Universal Robots PolyScope program: marco_robot_test.urp

Program marco_robot_test (installation=default directory=/programs createdIn=5.11.9.1010452 lastSavedIn=5.11.9.1010452 robotSerialNumber=20225200364)
Calibrated DH parameters: a=[0.00002, -0.569483, -0.54992, -0.00001, -0.000036, 0]; d=[0.180894, -146.691669, 192.918669, -46.053088, 0.119778, 0.115602]; alpha=[1.571425, -0.001534, 0.003359, 1.568739, -1.571477, 0]; deltaTheta=[0, 0.376258, -0.101074, -0.275185, -0.000002, 0]
Robot Program (runOnlyOnce=true)
  Script file /programs/usbdisk/marco_robot_5.script
    | def Machining3():
    |   # Default parameters:
    |   global speed_ms = 0.3
    |   global speed_rads = 0.75
    |   global accel_mss = 3
    |   global accel_radss = 1.2
    |   global blend_radius_m = 0.001
    | 
    |   # Add subprograms here
    |   # Start of main program
    |   # Program generated by RoboDK v5.6.5 for UR10e on 17/10/2023 12:20:24
    |   # Using nominal kinematics.
    |   blend_radius_m = 0.001
    |   speed_ms = 1.000
    |   # set_reference(p[0.335000, -0.154000, -0.002000, 0.000000, 0.000000, 0.000000])
    |   set_tcp(p[0.000000, 0.000000, 0.252000, 0.000000, 0.000000, 0.000000])
    |   # Show Tool
    |   movej([0.089160, -1.181798, -2.545827, -0.984764, 1.570796, 1.659956],accel_radss,speed_rads,0,blend_radius_m)
    |   movel([0.089160, -1.275562, -2.606033, -0.830794, 1.570796, 1.659956],accel_mss,speed_ms,0,blend_radius_m)
    |   speed_ms = 0.005
    |   movel([0.089160, -1.286495, -2.611612, -0.814282, 1.570796, 1.659956],accel_mss,speed_ms,0,blend_radius_m)
    |   movel([0.089160, -1.309264, -2.622500, -0.780625, 1.570796, 1.659956],accel_mss,speed_ms,0,blend_radius_m)
    |   movel([0.083541, -1.305906, -2.624527, -0.781955, 1.570796, 1.654337],accel_mss,speed_ms,0,blend_radius_m)
    |   movel([0.089160, -1.309264, -2.622500, -0.780625, 1.570796, 1.659956],accel_mss,speed_ms,0,blend_radius_m)
    |   movel([0.089160, -1.286495, -2.611612, -0.814282, 1.570796, 1.659956],accel_mss,speed_ms,0,blend_radius_m)
    |   movel([0.081204, -1.281682, -2.614420, -0.816287, 1.570796, 1.652001],accel_mss,speed_ms,0,blend_radius_m)
    |   movel([0.081204, -1.304518, -2.625361, -0.782510, 1.570796, 1.652001],accel_mss,speed_ms,0,blend_radius_m)
    |   movel([0.098719, -1.298708, -2.628824, -0.784857, 1.570796, 1.669516],accel_mss,speed_ms,0,blend_radius_m)
    |   movel([0.097011, -1.314060, -2.619578, -0.778751, 1.570796, 1.667807],accel_mss,speed_ms,0,blend_radius_m)
    |   movel([0.079808, -1.319640, -2.616140, -0.776609, 1.570796, 1.650604],accel_mss,speed_ms,0,blend_radius_m)
    |   movel([0.081204, -1.304518, -2.625361, -0.782510, 1.570796, 1.652001],accel_mss,speed_ms,0,blend_radius_m)
    |   movel([0.098719, -1.298708, -2.628824, -0.784857, 1.570796, 1.669516],accel_mss,speed_ms,0,blend_radius_m)
    |   movel([0.097011, -1.314060, -2.619578, -0.778751, 1.570796, 1.667807],accel_mss,speed_ms,0,blend_radius_m)
    |   movel([0.079808, -1.319640, -2.616140, -0.776609, 1.570796, 1.650604],accel_mss,speed_ms,0,blend_radius_m)
    |   movel([0.081204, -1.304518, -2.625361, -0.782510, 1.570796, 1.652001],accel_mss,speed_ms,0,blend_radius_m)
    |   movel([0.081204, -1.281682, -2.614420, -0.816287, 1.570796, 1.652001],accel_mss,speed_ms,0,blend_radius_m)
    |   movel([0.077108, -1.278531, -2.616242, -0.817615, 1.570796, 1.647904],accel_mss,speed_ms,0,blend_radius_m)
    |   movel([0.077108, -1.301410, -2.627219, -0.783760, 1.570796, 1.647904],accel_mss,speed_ms,0,blend_radius_m)
    |   movel([0.055264, -1.309051, -2.622629, -0.780709, 1.570796, 1.626060],accel_mss,speed_ms,0,blend_radius_m)
    |   movel([0.054551, -1.320244, -2.615765, -0.776379, 1.570796, 1.625347],accel_mss,speed_ms,0,blend_radius_m)
    |   movel([0.076104, -1.312829, -2.620331, -0.779229, 1.570796, 1.646901],accel_mss,speed_ms,0,blend_radius_m)
    |   movel([0.054551, -1.320244, -2.615765, -0.776379, 1.570796, 1.625347],accel_mss,speed_ms,0,blend_radius_m)
    |   movel([0.055264, -1.309051, -2.622629, -0.780709, 1.570796, 1.626060],accel_mss,speed_ms,0,blend_radius_m)
    |   movel([0.077108, -1.301410, -2.627219, -0.783760, 1.570796, 1.647904],accel_mss,speed_ms,0,blend_radius_m)
    |   movel([0.077108, -1.278531, -2.616242, -0.817615, 1.570796, 1.647904],accel_mss,speed_ms,0,blend_radius_m)
    |   movel([0.074534, -1.291116, -2.608888, -0.812385, 1.570796, 1.645331],accel_mss,speed_ms,0,blend_radius_m)
    |   movel([0.074534, -1.313820, -2.619725, -0.778844, 1.570796, 1.645331],accel_mss,speed_ms,0,blend_radius_m)
    |   movel([0.056039, -1.320179, -2.615806, -0.776404, 1.570796, 1.626835],accel_mss,speed_ms,0,blend_radius_m)
    |   movel([0.074534, -1.313820, -2.619725, -0.778844, 1.570796, 1.645331],accel_mss,speed_ms,0,blend_radius_m)
    |   movel([0.074534, -1.291116, -2.608888, -0.812385, 1.570796, 1.645331],accel_mss,speed_ms,0,blend_radius_m)
    |   movel([0.055828, -1.300854, -2.603061, -0.808474, 1.570796, 1.626625],accel_mss,speed_ms,0,blend_radius_m)
    |   movel([0.055828, -1.323418, -2.613789, -0.775182, 1.570796, 1.626625],accel_mss,speed_ms,0,blend_radius_m)
    |   movel([0.074252, -1.317114, -2.617702, -0.777573, 1.570796, 1.645049],accel_mss,speed_ms,0,blend_radius_m)
    |   movel([0.055828, -1.323418, -2.613789, -0.775182, 1.570796, 1.626625],accel_mss,speed_ms,0,blend_radius_m)
    |   movel([0.055828, -1.300854, -2.603061, -0.808474, 1.570796, 1.626625],accel_mss,speed_ms,0,blend_radius_m)
    |   movel([0.075501, -1.297125, -2.605307, -0.809958, 1.570796, 1.646297],accel_mss,speed_ms,0,blend_radius_m)
    |   movel([0.075501, -1.319743, -2.616077, -0.776570, 1.570796, 1.646297],accel_mss,speed_ms,0,blend_radius_m)
    |   movel([0.054122, -1.327025, -2.611526, -0.773837, 1.570796, 1.624918],accel_mss,speed_ms,0,blend_radius_m)
    |   movel([0.052635, -1.350841, -2.596143, -0.765405, 1.570796, 1.623432],accel_mss,speed_ms,0,blend_radius_m)
    |   movel([0.073235, -1.346070, -2.599287, -0.767032, 1.570796, 1.644031],accel_mss,speed_ms,0,blend_radius_m)
    |   movel([0.052635, -1.350841, -2.596143, -0.765405, 1.570796, 1.623432],accel_mss,speed_ms,0,blend_radius_m)
    |   movel([0.054122, -1.327025, -2.611526, -0.773837, 1.570796, 1.624918],accel_mss,speed_ms,0,blend_radius_m)
    |   movel([0.075501, -1.319743, -2.616077, -0.776570, 1.570796, 1.646297],accel_mss,speed_ms,0,blend_radius_m)
    |   movel([0.075501, -1.297125, -2.605307, -0.809958, 1.570796, 1.646297],accel_mss,speed_ms,0,blend_radius_m)
    |   movel([0.084967, -1.313702, -2.595186, -0.803501, 1.570796, 1.655763],accel_mss,speed_ms,0,blend_radius_m)
    |   movel([0.084967, -1.336075, -2.605773, -0.770542, 1.570796, 1.655763],accel_mss,speed_ms,0,blend_radius_m)
    |   movel([0.126975, -1.323371, -2.613818, -0.775199, 1.570796, 1.697771],accel_mss,speed_ms,0,blend_radius_m)
    |   movel([0.124703, -1.339286, -2.603704, -0.769399, 1.570796, 1.695499],accel_mss,speed_ms,0,blend_radius_m)
    |   movel([0.083467, -1.351474, -2.595724, -0.765192, 1.570796, 1.654263],accel_mss,speed_ms,0,blend_radius_m)
    |   movel([0.084967, -1.336075, -2.605773, -0.770542, 1.570796, 1.655763],accel_mss,speed_ms,0,blend_radius_m)
    |   movel([0.126975, -1.323371, -2.613818, -0.775199, 1.570796, 1.697771],accel_mss,speed_ms,0,blend_radius_m)
    |   movel([0.124703, -1.339286, -2.603704, -0.769399, 1.570796, 1.695499],accel_mss,speed_ms,0,blend_radius_m)
    |   movel([0.083467, -1.351474, -2.595724, -0.765192, 1.570796, 1.654263],accel_mss,speed_ms,0,blend_radius_m)
    |   movel([0.084967, -1.336075, -2.605773, -0.770542, 1.570796, 1.655763],accel_mss,speed_ms,0,blend_radius_m)
    |   movel([0.084967, -1.313702, -2.595186, -0.803501, 1.570796, 1.655763],accel_mss,speed_ms,0,blend_radius_m)
    |   movel([0.093012, -1.328943, -2.585565, -0.797880, 1.570796, 1.663809],accel_mss,speed_ms,0,blend_radius_m)
    |   movel([0.093012, -1.351081, -2.595984, -0.765324, 1.570796, 1.663809],accel_mss,speed_ms,0,blend_radius_m)
    |   movel([0.114947, -1.344626, -2.600233, -0.767530, 1.570796, 1.685744],accel_mss,speed_ms,0,blend_radius_m)
    |   movel([0.114417, -1.348663, -2.597583, -0.766144, 1.570796, 1.685214],accel_mss,speed_ms,0,blend_radius_m)
    |   movel([0.092587, -1.355051, -2.593343, -0.763996, 1.570796, 1.663383],accel_mss,speed_ms,0,blend_radius_m)
    |   movel([0.093012, -1.351081, -2.595984, -0.765324, 1.570796, 1.663809],accel_mss,speed_ms,0,blend_radius_m)
    |   movel([0.114947, -1.344626, -2.600233, -0.767530, 1.570796, 1.685744],accel_mss,speed_ms,0,blend_radius_m)
    |   movel([0.114417, -1.348663, -2.597583, -0.766144, 1.570796, 1.685214],accel_mss,speed_ms,0,blend_radius_m)
    |   movel([0.092587, -1.355051, -2.593343, -0.763996, 1.570796, 1.663383],accel_mss,speed_ms,0,blend_radius_m)
    |   movel([0.093012, -1.351081, -2.595984, -0.765324, 1.570796, 1.663809],accel_mss,speed_ms,0,blend_radius_m)
    |   movel([0.093012, -1.328943, -2.585565, -0.797880, 1.570796, 1.663809],accel_mss,speed_ms,0,blend_radius_m)
    |   movel([0.097348, -1.351902, -2.570489, -0.789998, 1.570796, 1.668144],accel_mss,speed_ms,0,blend_radius_m)
    |   movel([0.097348, -1.373670, -2.580657, -0.758062, 1.570796, 1.668144],accel_mss,speed_ms,0,blend_radius_m)
    |   movel([0.101037, -1.372618, -2.581387, -0.758385, 1.570796, 1.671834],accel_mss,speed_ms,0,blend_radius_m)
    |   movel([0.104717, -1.371577, -2.582107, -0.758705, 1.570796, 1.675514],accel_mss,speed_ms,0,blend_radius_m)
    |   movel([0.100259, -1.379284, -2.576735, -0.756370, 1.570796, 1.671055],accel_mss,speed_ms,0,blend_radius_m)
    |   movel([0.097348, -1.373670, -2.580657, -0.758062, 1.570796, 1.668144],accel_mss,speed_ms,0,blend_radius_m)
    |   movel([0.101037, -1.372618, -2.581387, -0.758385, 1.570796, 1.671834],accel_mss,speed_ms,0,blend_radius_m)
    |   movel([0.104717, -1.371577, -2.582107, -0.758705, 1.570796, 1.675514],accel_mss,speed_ms,0,blend_radius_m)
    |   movel([0.100259, -1.379284, -2.576735, -0.756370, 1.570796, 1.671055],accel_mss,speed_ms,0,blend_radius_m)
    |   movel([0.097348, -1.373670, -2.580657, -0.758062, 1.570796, 1.668144],accel_mss,speed_ms,0,blend_radius_m)
    |   movel([0.097348, -1.351902, -2.570489, -0.789998, 1.570796, 1.668144],accel_mss,speed_ms,0,blend_radius_m)
    |   movel([0.088027, -1.372703, -2.556208, -0.783478, 1.570796, 1.658823],accel_mss,speed_ms,0,blend_radius_m)
    |   movel([0.088027, -1.394119, -2.566152, -0.752118, 1.570796, 1.658823],accel_mss,speed_ms,0,blend_radius_m)
    |   movel([0.109776, -1.388105, -2.570480, -0.753803, 1.570796, 1.680572],accel_mss,speed_ms,0,blend_radius_m)
    |   movel([0.109257, -1.392184, -2.567551, -0.752654, 1.570796, 1.680053],accel_mss,speed_ms,0,blend_radius_m)
    |   movel([0.087614, -1.398134, -2.563233, -0.751022, 1.570796, 1.658410],accel_mss,speed_ms,0,blend_radius_m)
    |   movel([0.088027, -1.394119, -2.566152, -0.752118, 1.570796, 1.658823],accel_mss,speed_ms,0,blend_radius_m)
    |   movel([0.109776, -1.388105, -2.570480, -0.753803, 1.570796, 1.680572],accel_mss,speed_ms,0,blend_radius_m)
    |   movel([0.109257, -1.392184, -2.567551, -0.752654, 1.570796, 1.680053],accel_mss,speed_ms,0,blend_radius_m)
    |   movel([0.087614, -1.398134, -2.563233, -0.751022, 1.570796, 1.658410],accel_mss,speed_ms,0,blend_radius_m)
    |   movel([0.088027, -1.394119, -2.566152, -0.752118, 1.570796, 1.658823],accel_mss,speed_ms,0,blend_radius_m)
    |   movel([0.088027, -1.372703, -2.556208, -0.783478, 1.570796, 1.658823],accel_mss,speed_ms,0,blend_radius_m)
    |   movel([0.137771, -1.304245, -2.601003, -0.807141, 1.570796, 1.708567],accel_mss,speed_ms,0,blend_radius_m)
    |   movel([0.137771, -1.326759, -2.611694, -0.773936, 1.570796, 1.708567],accel_mss,speed_ms,0,blend_radius_m)
    |   movel([0.159338, -1.318850, -2.616630, -0.776910, 1.570796, 1.730135],accel_mss,speed_ms,0,blend_radius_m)
    |   movel([0.164004, -1.292855, -2.632269, -0.787265, 1.570796, 1.734800],accel_mss,speed_ms,0,blend_radius_m)
    |   movel([0.142128, -1.298999, -2.628652, -0.784738, 1.570796, 1.712924],accel_mss,speed_ms,0,blend_radius_m)
    |   movel([0.164004, -1.292855, -2.632269, -0.787265, 1.570796, 1.734800],accel_mss,speed_ms,0,blend_radius_m)
    |   movel([0.159338, -1.318850, -2.616630, -0.776910, 1.570796, 1.730135],accel_mss,speed_ms,0,blend_radius_m)
    |   movel([0.137771, -1.326759, -2.611694, -0.773936, 1.570796, 1.708567],accel_mss,speed_ms,0,blend_radius_m)
    |   movel([0.137771, -1.304245, -2.601003, -0.807141, 1.570796, 1.708567],accel_mss,speed_ms,0,blend_radius_m)
    |   movel([0.144204, -1.272270, -2.619828, -0.820291, 1.570796, 1.715001],accel_mss,speed_ms,0,blend_radius_m)
    |   movel([0.144204, -1.295233, -2.630875, -0.786282, 1.570796, 1.715001],accel_mss,speed_ms,0,blend_radius_m)
    |   movel([0.163060, -1.289910, -2.633985, -0.788494, 1.570796, 1.733856],accel_mss,speed_ms,0,blend_radius_m)
    |   movel([0.144204, -1.295233, -2.630875, -0.786282, 1.570796, 1.715001],accel_mss,speed_ms,0,blend_radius_m)
    |   movel([0.144204, -1.272270, -2.619828, -0.820291, 1.570796, 1.715001],accel_mss,speed_ms,0,blend_radius_m)
    |   movel([0.143289, -1.268681, -2.621861, -0.821846, 1.570796, 1.714086],accel_mss,speed_ms,0,blend_radius_m)
    |   movel([0.143289, -1.291691, -2.632948, -0.787749, 1.570796, 1.714086],accel_mss,speed_ms,0,blend_radius_m)
    |   movel([0.165352, -1.285426, -2.636577, -0.790386, 1.570796, 1.736149],accel_mss,speed_ms,0,blend_radius_m)
    |   movel([0.167598, -1.273136, -2.643552, -0.795701, 1.570796, 1.738395],accel_mss,speed_ms,0,blend_radius_m)
    |   movel([0.145223, -1.279606, -2.639904, -0.792879, 1.570796, 1.716019],accel_mss,speed_ms,0,blend_radius_m)
    |   movel([0.167598, -1.273136, -2.643552, -0.795701, 1.570796, 1.738395],accel_mss,speed_ms,0,blend_radius_m)
    |   movel([0.165352, -1.285426, -2.636577, -0.790386, 1.570796, 1.736149],accel_mss,speed_ms,0,blend_radius_m)
    |   movel([0.143289, -1.291691, -2.632948, -0.787749, 1.570796, 1.714086],accel_mss,speed_ms,0,blend_radius_m)
    |   movel([0.143289, -1.268681, -2.621861, -0.821846, 1.570796, 1.714086],accel_mss,speed_ms,0,blend_radius_m)
    |   movel([0.144765, -1.268733, -2.621832, -0.821824, 1.570796, 1.715562],accel_mss,speed_ms,0,blend_radius_m)
    |   movel([0.144765, -1.291742, -2.632919, -0.787728, 1.570796, 1.715562],accel_mss,speed_ms,0,blend_radius_m)
    |   movel([0.163697, -1.286370, -2.636034, -0.789985, 1.570796, 1.734494],accel_mss,speed_ms,0,blend_radius_m)
    |   movel([0.144765, -1.291742, -2.632919, -0.787728, 1.570796, 1.715562],accel_mss,speed_ms,0,blend_radius_m)
    |   movel([0.144765, -1.268733, -2.621832, -0.821824, 1.570796, 1.715562],accel_mss,speed_ms,0,blend_radius_m)
    |   movel([0.125413, -1.167058, -2.673236, -0.872095, 1.570796, 1.696210],accel_mss,speed_ms,0,blend_radius_m)
    |   movel([0.125413, -1.191107, -2.685463, -0.835818, 1.570796, 1.696210],accel_mss,speed_ms,0,blend_radius_m)
    |   movel([0.125706, -1.190153, -2.685906, -0.836330, 1.570796, 1.696503],accel_mss,speed_ms,0,blend_radius_m)
    |   movel([0.127514, -1.187943, -2.686927, -0.837519, 1.570796, 1.698310],accel_mss,speed_ms,0,blend_radius_m)
    |   movel([0.128757, -1.187262, -2.687241, -0.837886, 1.570796, 1.699553],accel_mss,speed_ms,0,blend_radius_m)
    |   movel([0.159607, -1.176201, -2.692265, -0.843923, 1.570796, 1.730403],accel_mss,speed_ms,0,blend_radius_m)
    |   movel([0.160858, -1.176036, -2.692339, -0.844014, 1.570796, 1.731655],accel_mss,speed_ms,0,blend_radius_m)
    |   movel([0.162120, -1.177291, -2.691776, -0.843322, 1.570796, 1.732916],accel_mss,speed_ms,0,blend_radius_m)
    |   movel([0.162101, -1.178007, -2.691454, -0.842928, 1.570796, 1.732898],accel_mss,speed_ms,0,blend_radius_m)
    |   movel([0.160218, -1.189028, -2.686427, -0.836935, 1.570796, 1.731014],accel_mss,speed_ms,0,blend_radius_m)
    |   movel([0.159776, -1.190238, -2.685867, -0.836284, 1.570796, 1.730573],accel_mss,speed_ms,0,blend_radius_m)
    |   movel([0.158190, -1.192057, -2.685022, -0.835310, 1.570796, 1.728986],accel_mss,speed_ms,0,blend_radius_m)
    |   movel([0.156814, -1.192816, -2.684669, -0.834905, 1.570796, 1.727611],accel_mss,speed_ms,0,blend_radius_m)
    |   movel([0.126529, -1.203419, -2.679664, -0.829306, 1.570796, 1.697325],accel_mss,speed_ms,0,blend_radius_m)
    |   movel([0.125786, -1.203591, -2.679582, -0.829216, 1.570796, 1.696582],accel_mss,speed_ms,0,blend_radius_m)
    |   movel([0.124122, -1.202858, -2.679932, -0.829599, 1.570796, 1.694918],accel_mss,speed_ms,0,blend_radius_m)
    |   movel([0.123975, -1.201767, -2.680452, -0.830170, 1.570796, 1.694771],accel_mss,speed_ms,0,blend_radius_m)
    |   movel([0.125413, -1.191107, -2.685463, -0.835818, 1.570796, 1.696210],accel_mss,speed_ms,0,blend_radius_m)
    |   movel([0.125706, -1.190153, -2.685906, -0.836330, 1.570796, 1.696503],accel_mss,speed_ms,0,blend_radius_m)
    |   movel([0.127514, -1.187943, -2.686927, -0.837519, 1.570796, 1.698310],accel_mss,speed_ms,0,blend_radius_m)
    |   movel([0.128757, -1.187262, -2.687241, -0.837886, 1.570796, 1.699553],accel_mss,speed_ms,0,blend_radius_m)
    |   movel([0.159607, -1.176201, -2.692265, -0.843923, 1.570796, 1.730403],accel_mss,speed_ms,0,blend_radius_m)
    |   movel([0.160858, -1.176036, -2.692339, -0.844014, 1.570796, 1.731655],accel_mss,speed_ms,0,blend_radius_m)
    |   movel([0.162120, -1.177291, -2.691776, -0.843322, 1.570796, 1.732916],accel_mss,speed_ms,0,blend_radius_m)
    |   movel([0.162101, -1.178007, -2.691454, -0.842928, 1.570796, 1.732898],accel_mss,speed_ms,0,blend_radius_m)
    |   movel([0.160218, -1.189028, -2.686427, -0.836935, 1.570796, 1.731014],accel_mss,speed_ms,0,blend_radius_m)
    |   movel([0.159776, -1.190238, -2.685867, -0.836284, 1.570796, 1.730573],accel_mss,speed_ms,0,blend_radius_m)
    |   movel([0.158190, -1.192057, -2.685022, -0.835310, 1.570796, 1.728986],accel_mss,speed_ms,0,blend_radius_m)
    |   movel([0.156814, -1.192816, -2.684669, -0.834905, 1.570796, 1.727611],accel_mss,speed_ms,0,blend_radius_m)
    |   movel([0.126529, -1.203419, -2.679664, -0.829306, 1.570796, 1.697325],accel_mss,speed_ms,0,blend_radius_m)
    |   movel([0.125786, -1.203591, -2.679582, -0.829216, 1.570796, 1.696582],accel_mss,speed_ms,0,blend_radius_m)
    |   movel([0.124122, -1.202858, -2.679932, -0.829599, 1.570796, 1.694918],accel_mss,speed_ms,0,blend_radius_m)
    |   movel([0.123975, -1.201767, -2.680452, -0.830170, 1.570796, 1.694771],accel_mss,speed_ms,0,blend_radius_m)
    |   movel([0.125413, -1.191107, -2.685463, -0.835818, 1.570796, 1.696210],accel_mss,speed_ms,0,blend_radius_m)
    |   movel([0.125413, -1.167058, -2.673236, -0.872095, 1.570796, 1.696210],accel_mss,speed_ms,0,blend_radius_m)
    |   movel([0.123336, -1.182593, -2.666121, -0.863674, 1.570796, 1.694132],accel_mss,speed_ms,0,blend_radius_m)
    |   movel([0.123336, -1.206525, -2.678175, -0.827689, 1.570796, 1.694132],accel_mss,speed_ms,0,blend_radius_m)
    |   movel([0.159381, -1.193945, -2.684142, -0.834303, 1.570796, 1.730178],accel_mss,speed_ms,0,blend_radius_m)
    |   movel([0.154982, -1.220061, -2.671558, -0.820770, 1.570796, 1.725778],accel_mss,speed_ms,0,blend_radius_m)
    |   movel([0.119973, -1.231829, -2.665636, -0.814924, 1.570796, 1.690769],accel_mss,speed_ms,0,blend_radius_m)
    |   movel([0.123336, -1.206525, -2.678175, -0.827689, 1.570796, 1.694132],accel_mss,speed_ms,0,blend_radius_m)
    |   movel([0.159381, -1.193945, -2.684142, -0.834303, 1.570796, 1.730178],accel_mss,speed_ms,0,blend_radius_m)
    |   movel([0.154982, -1.220061, -2.671558, -0.820770, 1.570796, 1.725778],accel_mss,speed_ms,0,blend_radius_m)
    |   movel([0.119973, -1.231829, -2.665636, -0.814924, 1.570796, 1.690769],accel_mss,speed_ms,0,blend_radius_m)
    |   movel([0.123336, -1.206525, -2.678175, -0.827689, 1.570796, 1.694132],accel_mss,speed_ms,0,blend_radius_m)
    |   movel([0.123336, -1.182593, -2.666121, -0.863674, 1.570796, 1.694132],accel_mss,speed_ms,0,blend_radius_m)
    |   movel([0.122335, -1.208273, -2.653796, -0.850320, 1.570796, 1.693131],accel_mss,speed_ms,0,blend_radius_m)
    |   movel([0.122335, -1.231976, -2.665561, -0.814852, 1.570796, 1.693131],accel_mss,speed_ms,0,blend_radius_m)
    |   movel([0.151945, -1.222034, -2.670576, -0.819779, 1.570796, 1.722741],accel_mss,speed_ms,0,blend_radius_m)
    |   movel([0.153970, -1.222028, -2.670579, -0.819782, 1.570796, 1.724766],accel_mss,speed_ms,0,blend_radius_m)
    |   movel([0.154423, -1.223410, -2.669889, -0.819090, 1.570796, 1.725219],accel_mss,speed_ms,0,blend_radius_m)
    |   movel([0.153408, -1.225329, -2.668927, -0.818133, 1.570796, 1.724204],accel_mss,speed_ms,0,blend_radius_m)
    |   movel([0.151526, -1.226585, -2.668295, -0.817510, 1.570796, 1.722322],accel_mss,speed_ms,0,blend_radius_m)
    |   movel([0.121726, -1.236519, -2.663231, -0.812639, 1.570796, 1.692523],accel_mss,speed_ms,0,blend_radius_m)
    |   movel([0.120074, -1.236452, -2.663266, -0.812672, 1.570796, 1.690871],accel_mss,speed_ms,0,blend_radius_m)
    |   movel([0.119542, -1.235104, -2.663959, -0.813326, 1.570796, 1.690338],accel_mss,speed_ms,0,blend_radius_m)
    |   movel([0.120485, -1.233242, -2.664914, -0.814233, 1.570796, 1.691281],accel_mss,speed_ms,0,blend_radius_m)
    |   movel([0.122335, -1.231976, -2.665561, -0.814852, 1.570796, 1.693131],accel_mss,speed_ms,0,blend_radius_m)
    |   movel([0.151945, -1.222034, -2.670576, -0.819779, 1.570796, 1.722741],accel_mss,speed_ms,0,blend_radius_m)
    |   movel([0.153970, -1.222028, -2.670579, -0.819782, 1.570796, 1.724766],accel_mss,speed_ms,0,blend_radius_m)
    |   movel([0.154423, -1.223410, -2.669889, -0.819090, 1.570796, 1.725219],accel_mss,speed_ms,0,blend_radius_m)
    |   movel([0.153408, -1.225329, -2.668927, -0.818133, 1.570796, 1.724204],accel_mss,speed_ms,0,blend_radius_m)
    |   movel([0.151526, -1.226585, -2.668295, -0.817510, 1.570796, 1.722322],accel_mss,speed_ms,0,blend_radius_m)
    |   movel([0.121726, -1.236519, -2.663231, -0.812639, 1.570796, 1.692523],accel_mss,speed_ms,0,blend_radius_m)
    |   movel([0.120074, -1.236452, -2.663266, -0.812672, 1.570796, 1.690871],accel_mss,speed_ms,0,blend_radius_m)
    |   movel([0.119542, -1.235104, -2.663959, -0.813326, 1.570796, 1.690338],accel_mss,speed_ms,0,blend_radius_m)
    |   movel([0.120485, -1.233242, -2.664914, -0.814233, 1.570796, 1.691281],accel_mss,speed_ms,0,blend_radius_m)
    |   movel([0.122335, -1.231976, -2.665561, -0.814852, 1.570796, 1.693131],accel_mss,speed_ms,0,blend_radius_m)
    |   movel([0.122335, -1.208273, -2.653796, -0.850320, 1.570796, 1.693131],accel_mss,speed_ms,0,blend_radius_m)
    |   movel([0.121590, -1.213891, -2.651003, -0.847495, 1.570796, 1.692386],accel_mss,speed_ms,0,blend_radius_m)
    |   movel([0.121590, -1.237538, -2.662705, -0.812146, 1.570796, 1.692386],accel_mss,speed_ms,0,blend_radius_m)
    |   movel([0.151010, -1.227741, -2.667711, -0.816937, 1.570796, 1.721806],accel_mss,speed_ms,0,blend_radius_m)
    |   movel([0.153022, -1.227740, -2.667712, -0.816937, 1.570796, 1.723819],accel_mss,speed_ms,0,blend_radius_m)
    |   movel([0.153474, -1.229110, -2.667018, -0.816260, 1.570796, 1.724271],accel_mss,speed_ms,0,blend_radius_m)
    |   movel([0.152465, -1.231024, -2.666046, -0.815319, 1.570796, 1.723261],accel_mss,speed_ms,0,blend_radius_m)
    |   movel([0.150598, -1.232252, -2.665420, -0.814717, 1.570796, 1.721394],accel_mss,speed_ms,0,blend_radius_m)
    |   movel([0.120989, -1.242042, -2.660366, -0.809981, 1.570796, 1.691785],accel_mss,speed_ms,0,blend_radius_m)
    |   movel([0.119345, -1.241985, -2.660395, -0.810008, 1.570796, 1.690141],accel_mss,speed_ms,0,blend_radius_m)
    |   movel([0.118816, -1.240634, -2.661100, -0.810655, 1.570796, 1.689612],accel_mss,speed_ms,0,blend_radius_m)
    |   movel([0.119752, -1.238790, -2.662057, -0.811542, 1.570796, 1.690548],accel_mss,speed_ms,0,blend_radius_m)
    |   movel([0.121590, -1.237538, -2.662705, -0.812146, 1.570796, 1.692386],accel_mss,speed_ms,0,blend_radius_m)
    |   movel([0.151010, -1.227741, -2.667711, -0.816937, 1.570796, 1.721806],accel_mss,speed_ms,0,blend_radius_m)
    |   movel([0.153022, -1.227740, -2.667712, -0.816937, 1.570796, 1.723819],accel_mss,speed_ms,0,blend_radius_m)
    |   movel([0.153474, -1.229110, -2.667018, -0.816260, 1.570796, 1.724271],accel_mss,speed_ms,0,blend_radius_m)
    |   movel([0.152465, -1.231024, -2.666046, -0.815319, 1.570796, 1.723261],accel_mss,speed_ms,0,blend_radius_m)
    |   movel([0.150598, -1.232252, -2.665420, -0.814717, 1.570796, 1.721394],accel_mss,speed_ms,0,blend_radius_m)
    |   movel([0.120989, -1.242042, -2.660366, -0.809981, 1.570796, 1.691785],accel_mss,speed_ms,0,blend_radius_m)
    |   movel([0.119345, -1.241985, -2.660395, -0.810008, 1.570796, 1.690141],accel_mss,speed_ms,0,blend_radius_m)
    |   movel([0.118816, -1.240634, -2.661100, -0.810655, 1.570796, 1.689612],accel_mss,speed_ms,0,blend_radius_m)
    |   movel([0.119752, -1.238790, -2.662057, -0.811542, 1.570796, 1.690548],accel_mss,speed_ms,0,blend_radius_m)
    |   movel([0.121590, -1.237538, -2.662705, -0.812146, 1.570796, 1.692386],accel_mss,speed_ms,0,blend_radius_m)
    |   movel([0.121590, -1.213891, -2.651003, -0.847495, 1.570796, 1.692386],accel_mss,speed_ms,0,blend_radius_m)
    |   movel([0.118388, -1.220324, -2.647761, -0.844303, 1.570796, 1.689184],accel_mss,speed_ms,0,blend_radius_m)
    |   movel([0.118388, -1.243905, -2.659391, -0.809093, 1.570796, 1.689184],accel_mss,speed_ms,0,blend_radius_m)
    |   movel([0.152910, -1.232509, -2.665289, -0.814591, 1.570796, 1.723707],accel_mss,speed_ms,0,blend_radius_m)
    |   movel([0.147205, -1.267322, -2.646785, -0.798282, 1.570796, 1.718001],accel_mss,speed_ms,0,blend_radius_m)
    |   movel([0.114019, -1.277736, -2.640964, -0.793690, 1.570796, 1.684815],accel_mss,speed_ms,0,blend_radius_m)
    |   movel([0.118388, -1.243905, -2.659391, -0.809093, 1.570796, 1.689184],accel_mss,speed_ms,0,blend_radius_m)
    |   movel([0.152910, -1.232509, -2.665289, -0.814591, 1.570796, 1.723707],accel_mss,speed_ms,0,blend_radius_m)
    |   movel([0.147205, -1.267322, -2.646785, -0.798282, 1.570796, 1.718001],accel_mss,speed_ms,0,blend_radius_m)
    |   movel([0.114019, -1.277736, -2.640964, -0.793690, 1.570796, 1.684815],accel_mss,speed_ms,0,blend_radius_m)
    |   movel([0.118388, -1.243905, -2.659391, -0.809093, 1.570796, 1.689184],accel_mss,speed_ms,0,blend_radius_m)
    |   movel([0.118388, -1.220324, -2.647761, -0.844303, 1.570796, 1.689184],accel_mss,speed_ms,0,blend_radius_m)
    |   movel([0.148123, -1.243372, -2.635760, -0.833257, 1.570796, 1.718919],accel_mss,speed_ms,0,blend_radius_m)
    |   movel([0.148123, -1.266696, -2.647131, -0.798562, 1.570796, 1.718919],accel_mss,speed_ms,0,blend_radius_m)
    |   movel([0.148538, -1.266484, -2.647248, -0.798657, 1.570796, 1.719334],accel_mss,speed_ms,0,blend_radius_m)
    |   movel([0.157718, -1.263743, -2.648755, -0.799891, 1.570796, 1.728514],accel_mss,speed_ms,0,blend_radius_m)
    |   movel([0.158038, -1.263698, -2.648780, -0.799911, 1.570796, 1.728835],accel_mss,speed_ms,0,blend_radius_m)
    |   movel([0.158373, -1.263888, -2.648676, -0.799825, 1.570796, 1.729169],accel_mss,speed_ms,0,blend_radius_m)
    |   movel([0.158443, -1.264268, -2.648467, -0.799654, 1.570796, 1.729239],accel_mss,speed_ms,0,blend_radius_m)
    |   movel([0.156589, -1.274995, -2.642509, -0.794885, 1.570796, 1.727385],accel_mss,speed_ms,0,blend_radius_m)
    |   movel([0.156411, -1.275404, -2.642279, -0.794706, 1.570796, 1.727207],accel_mss,speed_ms,0,blend_radius_m)
    |   movel([0.156020, -1.275800, -2.642056, -0.794533, 1.570796, 1.726817],accel_mss,speed_ms,0,blend_radius_m)
    |   movel([0.155609, -1.276005, -2.641940, -0.794443, 1.570796, 1.726405],accel_mss,speed_ms,0,blend_radius_m)
    |   movel([0.146557, -1.278660, -2.640441, -0.793289, 1.570796, 1.717354],accel_mss,speed_ms,0,blend_radius_m)
    |   movel([0.145878, -1.278457, -2.640555, -0.793376, 1.570796, 1.716674],accel_mss,speed_ms,0,blend_radius_m)
    |   movel([0.145847, -1.278148, -2.640730, -0.793511, 1.570796, 1.716644],accel_mss,speed_ms,0,blend_radius_m)
    |   movel([0.147569, -1.267511, -2.646681, -0.798197, 1.570796, 1.718365],accel_mss,speed_ms,0,blend_radius_m)
    |   movel([0.147672, -1.267206, -2.646850, -0.798334, 1.570796, 1.718469],accel_mss,speed_ms,0,blend_radius_m)
    |   movel([0.148123, -1.266696, -2.647131, -0.798562, 1.570796, 1.718919],accel_mss,speed_ms,0,blend_radius_m)
    |   movel([0.148538, -1.266484, -2.647248, -0.798657, 1.570796, 1.719334],accel_mss,speed_ms,0,blend_radius_m)
    |   movel([0.157718, -1.263743, -2.648755, -0.799891, 1.570796, 1.728514],accel_mss,speed_ms,0,blend_radius_m)
    |   movel([0.158038, -1.263698, -2.648780, -0.799911, 1.570796, 1.728835],accel_mss,speed_ms,0,blend_radius_m)
    |   movel([0.158373, -1.263888, -2.648676, -0.799825, 1.570796, 1.729169],accel_mss,speed_ms,0,blend_radius_m)
    |   movel([0.158443, -1.264268, -2.648467, -0.799654, 1.570796, 1.729239],accel_mss,speed_ms,0,blend_radius_m)
    |   movel([0.156589, -1.274995, -2.642509, -0.794885, 1.570796, 1.727385],accel_mss,speed_ms,0,blend_radius_m)
    |   movel([0.156411, -1.275404, -2.642279, -0.794706, 1.570796, 1.727207],accel_mss,speed_ms,0,blend_radius_m)
    |   movel([0.156020, -1.275800, -2.642056, -0.794533, 1.570796, 1.726817],accel_mss,speed_ms,0,blend_radius_m)
    |   movel([0.155609, -1.276005, -2.641940, -0.794443, 1.570796, 1.726405],accel_mss,speed_ms,0,blend_radius_m)
    |   movel([0.146557, -1.278660, -2.640441, -0.793289, 1.570796, 1.717354],accel_mss,speed_ms,0,blend_radius_m)
    |   movel([0.145878, -1.278457, -2.640555, -0.793376, 1.570796, 1.716674],accel_mss,speed_ms,0,blend_radius_m)
    |   movel([0.145847, -1.278148, -2.640730, -0.793511, 1.570796, 1.716644],accel_mss,speed_ms,0,blend_radius_m)
    |   movel([0.147569, -1.267511, -2.646681, -0.798197, 1.570796, 1.718365],accel_mss,speed_ms,0,blend_radius_m)
    |   movel([0.147672, -1.267206, -2.646850, -0.798334, 1.570796, 1.718469],accel_mss,speed_ms,0,blend_radius_m)
    |   movel([0.148123, -1.266696, -2.647131, -0.798562, 1.570796, 1.718919],accel_mss,speed_ms,0,blend_radius_m)
    |   movel([0.148123, -1.243372, -2.635760, -0.833257, 1.570796, 1.718919],accel_mss,speed_ms,0,blend_radius_m)
    |   movel([0.158944, -1.240765, -2.637148, -0.834476, 1.570796, 1.729740],accel_mss,speed_ms,0,blend_radius_m)
    |   movel([0.158944, -1.264120, -2.648548, -0.799720, 1.570796, 1.729740],accel_mss,speed_ms,0,blend_radius_m)
    |   movel([0.159066, -1.263809, -2.648719, -0.799861, 1.570796, 1.729863],accel_mss,speed_ms,0,blend_radius_m)
    |   movel([0.159522, -1.263298, -2.648999, -0.800092, 1.570796, 1.730319],accel_mss,speed_ms,0,blend_radius_m)
    |   movel([0.159940, -1.263088, -2.649114, -0.800187, 1.570796, 1.730736],accel_mss,speed_ms,0,blend_radius_m)
    |   movel([0.169139, -1.260415, -2.650573, -0.801401, 1.570796, 1.739936],accel_mss,speed_ms,0,blend_radius_m)
    |   movel([0.169445, -1.260377, -2.650593, -0.801418, 1.570796, 1.740242],accel_mss,speed_ms,0,blend_radius_m)
    |   movel([0.169791, -1.260568, -2.650489, -0.801331, 1.570796, 1.740587],accel_mss,speed_ms,0,blend_radius_m)
    |   movel([0.169841, -1.260957, -2.650278, -0.801154, 1.570796, 1.740638],accel_mss,speed_ms,0,blend_radius_m)
    |   movel([0.167848, -1.271777, -2.644311, -0.796301, 1.570796, 1.738644],accel_mss,speed_ms,0,blend_radius_m)
    |   movel([0.167665, -1.272188, -2.644082, -0.796119, 1.570796, 1.738461],accel_mss,speed_ms,0,blend_radius_m)
    |   movel([0.167284, -1.272581, -2.643862, -0.795946, 1.570796, 1.738080],accel_mss,speed_ms,0,blend_radius_m)
    |   movel([0.166870, -1.272784, -2.643749, -0.795856, 1.570796, 1.737667],accel_mss,speed_ms,0,blend_radius_m)
    |   movel([0.157800, -1.275372, -2.642297, -0.794720, 1.570796, 1.728596],accel_mss,speed_ms,0,blend_radius_m)
    |   movel([0.157125, -1.275160, -2.642416, -0.794813, 1.570796, 1.727921],accel_mss,speed_ms,0,blend_radius_m)
    |   movel([0.157084, -1.274852, -2.642590, -0.794948, 1.570796, 1.727880],accel_mss,speed_ms,0,blend_radius_m)
    |   movel([0.158944, -1.264120, -2.648548, -0.799720, 1.570796, 1.729740],accel_mss,speed_ms,0,blend_radius_m)
    |   movel([0.159066, -1.263809, -2.648719, -0.799861, 1.570796, 1.729863],accel_mss,speed_ms,0,blend_radius_m)
    |   movel([0.159522, -1.263298, -2.648999, -0.800092, 1.570796, 1.730319],accel_mss,speed_ms,0,blend_radius_m)
    |   movel([0.159940, -1.263088, -2.649114, -0.800187, 1.570796, 1.730736],accel_mss,speed_ms,0,blend_radius_m)
    |   movel([0.169139, -1.260415, -2.650573, -0.801401, 1.570796, 1.739936],accel_mss,speed_ms,0,blend_radius_m)
    |   movel([0.169445, -1.260377, -2.650593, -0.801418, 1.570796, 1.740242],accel_mss,speed_ms,0,blend_radius_m)
    |   movel([0.169791, -1.260568, -2.650489, -0.801331, 1.570796, 1.740587],accel_mss,speed_ms,0,blend_radius_m)
    |   movel([0.169841, -1.260957, -2.650278, -0.801154, 1.570796, 1.740638],accel_mss,speed_ms,0,blend_radius_m)
    |   movel([0.167848, -1.271777, -2.644311, -0.796301, 1.570796, 1.738644],accel_mss,speed_ms,0,blend_radius_m)
    |   movel([0.167665, -1.272188, -2.644082, -0.796119, 1.570796, 1.738461],accel_mss,speed_ms,0,blend_radius_m)
    |   movel([0.167284, -1.272581, -2.643862, -0.795946, 1.570796, 1.738080],accel_mss,speed_ms,0,blend_radius_m)
    |   movel([0.166870, -1.272784, -2.643749, -0.795856, 1.570796, 1.737667],accel_mss,speed_ms,0,blend_radius_m)
    |   movel([0.157800, -1.275372, -2.642297, -0.794720, 1.570796, 1.728596],accel_mss,speed_ms,0,blend_radius_m)
    |   movel([0.157125, -1.275160, -2.642416, -0.794813, 1.570796, 1.727921],accel_mss,speed_ms,0,blend_radius_m)
    |   movel([0.157084, -1.274852, -2.642590, -0.794948, 1.570796, 1.727880],accel_mss,speed_ms,0,blend_radius_m)
    |   movel([0.158944, -1.264120, -2.648548, -0.799720, 1.570796, 1.729740],accel_mss,speed_ms,0,blend_radius_m)
    |   movel([0.158944, -1.240765, -2.637148, -0.834476, 1.570796, 1.729740],accel_mss,speed_ms,0,blend_radius_m)
    |   movel([0.166870, -1.249533, -2.632447, -0.830409, 1.570796, 1.737667],accel_mss,speed_ms,0,blend_radius_m)
    |   movel([0.166870, -1.272784, -2.643749, -0.795856, 1.570796, 1.737667],accel_mss,speed_ms,0,blend_radius_m)
    |   movel([0.167284, -1.272581, -2.643862, -0.795946, 1.570796, 1.738080],accel_mss,speed_ms,0,blend_radius_m)
    |   movel([0.166870, -1.272784, -2.643749, -0.795856, 1.570796, 1.737667],accel_mss,speed_ms,0,blend_radius_m)
    |   movel([0.166870, -1.249533, -2.632447, -0.830409, 1.570796, 1.737667],accel_mss,speed_ms,0,blend_radius_m)
    |   movel([0.163697, -1.263290, -2.624886, -0.824212, 1.570796, 1.734494],accel_mss,speed_ms,0,blend_radius_m)
    |   movel([0.163697, -1.286370, -2.636034, -0.789985, 1.570796, 1.734494],accel_mss,speed_ms,0,blend_radius_m)
    |   movel([0.164641, -1.286424, -2.636002, -0.789962, 1.570796, 1.735438],accel_mss,speed_ms,0,blend_radius_m)
    |   movel([0.164999, -1.287368, -2.635458, -0.789563, 1.570796, 1.735796],accel_mss,speed_ms,0,blend_radius_m)
    |   movel([0.164276, -1.288585, -2.634754, -0.789050, 1.570796, 1.735073],accel_mss,speed_ms,0,blend_radius_m)
    |   movel([0.163183, -1.289224, -2.634383, -0.788782, 1.570796, 1.733980],accel_mss,speed_ms,0,blend_radius_m)
    |   movel([0.144313, -1.294556, -2.631272, -0.786561, 1.570796, 1.715109],accel_mss,speed_ms,0,blend_radius_m)
    |   movel([0.143344, -1.294502, -2.631304, -0.786583, 1.570796, 1.714140],accel_mss,speed_ms,0,blend_radius_m)
    |   movel([0.142985, -1.293602, -2.631832, -0.786956, 1.570796, 1.713782],accel_mss,speed_ms,0,blend_radius_m)
    |   movel([0.143713, -1.292360, -2.632558, -0.787471, 1.570796, 1.714509],accel_mss,speed_ms,0,blend_radius_m)
    |   movel([0.144765, -1.291742, -2.632919, -0.787728, 1.570796, 1.715562],accel_mss,speed_ms,0,blend_radius_m)
    |   movel([0.143713, -1.292360, -2.632558, -0.787471, 1.570796, 1.714509],accel_mss,speed_ms,0,blend_radius_m)
    |   movel([0.142985, -1.293602, -2.631832, -0.786956, 1.570796, 1.713782],accel_mss,speed_ms,0,blend_radius_m)
    |   movel([0.143344, -1.294502, -2.631304, -0.786583, 1.570796, 1.714140],accel_mss,speed_ms,0,blend_radius_m)
    |   movel([0.144313, -1.294556, -2.631272, -0.786561, 1.570796, 1.715109],accel_mss,speed_ms,0,blend_radius_m)
    |   movel([0.163183, -1.289224, -2.634383, -0.788782, 1.570796, 1.733980],accel_mss,speed_ms,0,blend_radius_m)
    |   movel([0.164276, -1.288585, -2.634754, -0.789050, 1.570796, 1.735073],accel_mss,speed_ms,0,blend_radius_m)
    |   movel([0.164999, -1.287368, -2.635458, -0.789563, 1.570796, 1.735796],accel_mss,speed_ms,0,blend_radius_m)
    |   movel([0.164641, -1.286424, -2.636002, -0.789962, 1.570796, 1.735438],accel_mss,speed_ms,0,blend_radius_m)
    |   movel([0.163697, -1.286370, -2.636034, -0.789985, 1.570796, 1.734494],accel_mss,speed_ms,0,blend_radius_m)
    |   movel([0.163697, -1.263290, -2.624886, -0.824212, 1.570796, 1.734494],accel_mss,speed_ms,0,blend_radius_m)
    |   movel([0.144204, -1.272270, -2.619828, -0.820291, 1.570796, 1.715001],accel_mss,speed_ms,0,blend_radius_m)
    |   movel([0.144204, -1.295233, -2.630875, -0.786282, 1.570796, 1.715001],accel_mss,speed_ms,0,blend_radius_m)
    |   movel([0.143154, -1.295859, -2.630507, -0.786024, 1.570796, 1.713951],accel_mss,speed_ms,0,blend_radius_m)
    |   movel([0.142432, -1.297080, -2.629786, -0.785522, 1.570796, 1.713229],accel_mss,speed_ms,0,blend_radius_m)
    |   movel([0.142790, -1.297976, -2.629257, -0.785155, 1.570796, 1.713587],accel_mss,speed_ms,0,blend_radius_m)
    |   movel([0.143756, -1.298031, -2.629225, -0.785133, 1.570796, 1.714552],accel_mss,speed_ms,0,blend_radius_m)
    |   movel([0.162550, -1.292749, -2.632331, -0.787309, 1.570796, 1.733346],accel_mss,speed_ms,0,blend_radius_m)
    |   movel([0.163638, -1.292114, -2.632702, -0.787574, 1.570796, 1.734434],accel_mss,speed_ms,0,blend_radius_m)
    |   movel([0.164357, -1.290905, -2.633407, -0.788078, 1.570796, 1.735154],accel_mss,speed_ms,0,blend_radius_m)
    |   movel([0.163998, -1.289978, -2.633946, -0.788465, 1.570796, 1.734794],accel_mss,speed_ms,0,blend_radius_m)
    |   movel([0.163060, -1.289910, -2.633985, -0.788494, 1.570796, 1.733856],accel_mss,speed_ms,0,blend_radius_m)
    |   movel([0.163998, -1.289978, -2.633946, -0.788465, 1.570796, 1.734794],accel_mss,speed_ms,0,blend_radius_m)
    |   movel([0.164357, -1.290905, -2.633407, -0.788078, 1.570796, 1.735154],accel_mss,speed_ms,0,blend_radius_m)
    |   movel([0.163638, -1.292114, -2.632702, -0.787574, 1.570796, 1.734434],accel_mss,speed_ms,0,blend_radius_m)
    |   movel([0.162550, -1.292749, -2.632331, -0.787309, 1.570796, 1.733346],accel_mss,speed_ms,0,blend_radius_m)
    |   movel([0.143756, -1.298031, -2.629225, -0.785133, 1.570796, 1.714552],accel_mss,speed_ms,0,blend_radius_m)
    |   movel([0.142790, -1.297976, -2.629257, -0.785155, 1.570796, 1.713587],accel_mss,speed_ms,0,blend_radius_m)
    |   movel([0.142432, -1.297080, -2.629786, -0.785522, 1.570796, 1.713229],accel_mss,speed_ms,0,blend_radius_m)
    |   movel([0.143154, -1.295859, -2.630507, -0.786024, 1.570796, 1.713951],accel_mss,speed_ms,0,blend_radius_m)
    |   movel([0.144204, -1.295233, -2.630875, -0.786282, 1.570796, 1.715001],accel_mss,speed_ms,0,blend_radius_m)
    |   movel([0.144204, -1.272270, -2.619828, -0.820291, 1.570796, 1.715001],accel_mss,speed_ms,0,blend_radius_m)
    |   movel([0.140763, -1.263908, -2.624542, -0.823939, 1.570796, 1.711559],accel_mss,speed_ms,0,blend_radius_m)
    |   movel([0.140763, -1.286980, -2.635682, -0.789727, 1.570796, 1.711559],accel_mss,speed_ms,0,blend_radius_m)
    |   movel([0.139826, -1.288717, -2.634677, -0.788994, 1.570796, 1.710622],accel_mss,speed_ms,0,blend_radius_m)
    |   movel([0.138100, -1.289807, -2.634045, -0.788537, 1.570796, 1.708896],accel_mss,speed_ms,0,blend_radius_m)
    |   movel([0.110362, -1.298317, -2.629056, -0.785016, 1.570796, 1.681158],accel_mss,speed_ms,0,blend_radius_m)
    |   movel([0.108814, -1.298239, -2.629102, -0.785048, 1.570796, 1.679611],accel_mss,speed_ms,0,blend_radius_m)
    |   movel([0.108301, -1.296993, -2.629838, -0.785558, 1.570796, 1.679097],accel_mss,speed_ms,0,blend_radius_m)
    |   movel([0.109145, -1.295335, -2.630815, -0.786240, 1.570796, 1.679941],accel_mss,speed_ms,0,blend_radius_m)
    |   movel([0.110874, -1.294213, -2.631474, -0.786703, 1.570796, 1.681670],accel_mss,speed_ms,0,blend_radius_m)
    |   movel([0.138424, -1.285706, -2.636416, -0.790267, 1.570796, 1.709221],accel_mss,speed_ms,0,blend_radius_m)
    |   movel([0.140319, -1.285721, -2.636407, -0.790260, 1.570796, 1.711115],accel_mss,speed_ms,0,blend_radius_m)
    |   movel([0.140763, -1.286980, -2.635682, -0.789727, 1.570796, 1.711559],accel_mss,speed_ms,0,blend_radius_m)
    |   movel([0.139826, -1.288717, -2.634677, -0.788994, 1.570796, 1.710622],accel_mss,speed_ms,0,blend_radius_m)
    |   movel([0.138100, -1.289807, -2.634045, -0.788537, 1.570796, 1.708896],accel_mss,speed_ms,0,blend_radius_m)
    |   movel([0.110362, -1.298317, -2.629056, -0.785016, 1.570796, 1.681158],accel_mss,speed_ms,0,blend_radius_m)
    |   movel([0.108814, -1.298239, -2.629102, -0.785048, 1.570796, 1.679611],accel_mss,speed_ms,0,blend_radius_m)
    |   movel([0.108301, -1.296993, -2.629838, -0.785558, 1.570796, 1.679097],accel_mss,speed_ms,0,blend_radius_m)
    |   movel([0.109145, -1.295335, -2.630815, -0.786240, 1.570796, 1.679941],accel_mss,speed_ms,0,blend_radius_m)
    |   movel([0.110874, -1.294213, -2.631474, -0.786703, 1.570796, 1.681670],accel_mss,speed_ms,0,blend_radius_m)
    |   movel([0.138424, -1.285706, -2.636416, -0.790267, 1.570796, 1.709221],accel_mss,speed_ms,0,blend_radius_m)
    |   movel([0.140319, -1.285721, -2.636407, -0.790260, 1.570796, 1.711115],accel_mss,speed_ms,0,blend_radius_m)
    |   movel([0.140763, -1.286980, -2.635682, -0.789727, 1.570796, 1.711559],accel_mss,speed_ms,0,blend_radius_m)
    |   movel([0.140763, -1.263908, -2.624542, -0.823939, 1.570796, 1.711559],accel_mss,speed_ms,0,blend_radius_m)
    |   movel([0.139542, -1.267692, -2.622419, -0.822278, 1.570796, 1.710338],accel_mss,speed_ms,0,blend_radius_m)
    |   movel([0.139542, -1.290714, -2.633517, -0.788157, 1.570796, 1.710338],accel_mss,speed_ms,0,blend_radius_m)
    |   movel([0.139985, -1.291964, -2.632789, -0.787636, 1.570796, 1.710781],accel_mss,speed_ms,0,blend_radius_m)
    |   movel([0.139056, -1.293674, -2.631789, -0.786925, 1.570796, 1.709853],accel_mss,speed_ms,0,blend_radius_m)
    |   movel([0.137339, -1.294766, -2.631149, -0.786474, 1.570796, 1.708135],accel_mss,speed_ms,0,blend_radius_m)
    |   movel([0.109759, -1.303165, -2.626171, -0.783052, 1.570796, 1.680555],accel_mss,speed_ms,0,blend_radius_m)
    |   movel([0.108221, -1.303073, -2.626226, -0.783089, 1.570796, 1.679018],accel_mss,speed_ms,0,blend_radius_m)
    |   movel([0.107708, -1.301848, -2.626958, -0.783583, 1.570796, 1.678505],accel_mss,speed_ms,0,blend_radius_m)
    |   movel([0.108548, -1.300191, -2.627945, -0.784254, 1.570796, 1.679345],accel_mss,speed_ms,0,blend_radius_m)
    |   movel([0.110267, -1.299080, -2.628604, -0.784705, 1.570796, 1.681063],accel_mss,speed_ms,0,blend_radius_m)
    |   movel([0.137660, -1.290683, -2.633535, -0.788170, 1.570796, 1.708456],accel_mss,speed_ms,0,blend_radius_m)
    |   movel([0.139542, -1.290714, -2.633517, -0.788157, 1.570796, 1.710338],accel_mss,speed_ms,0,blend_radius_m)
    |   movel([0.139985, -1.291964, -2.632789, -0.787636, 1.570796, 1.710781],accel_mss,speed_ms,0,blend_radius_m)
    |   movel([0.139056, -1.293674, -2.631789, -0.786925, 1.570796, 1.709853],accel_mss,speed_ms,0,blend_radius_m)
    |   movel([0.137339, -1.294766, -2.631149, -0.786474, 1.570796, 1.708135],accel_mss,speed_ms,0,blend_radius_m)
    |   movel([0.109759, -1.303165, -2.626171, -0.783052, 1.570796, 1.680555],accel_mss,speed_ms,0,blend_radius_m)
    |   movel([0.108221, -1.303073, -2.626226, -0.783089, 1.570796, 1.679018],accel_mss,speed_ms,0,blend_radius_m)
    |   movel([0.107708, -1.301848, -2.626958, -0.783583, 1.570796, 1.678505],accel_mss,speed_ms,0,blend_radius_m)
    |   movel([0.108548, -1.300191, -2.627945, -0.784254, 1.570796, 1.679345],accel_mss,speed_ms,0,blend_radius_m)
    |   movel([0.110267, -1.299080, -2.628604, -0.784705, 1.570796, 1.681063],accel_mss,speed_ms,0,blend_radius_m)
    |   movel([0.137660, -1.290683, -2.633535, -0.788170, 1.570796, 1.708456],accel_mss,speed_ms,0,blend_radius_m)
    |   movel([0.139542, -1.290714, -2.633517, -0.788157, 1.570796, 1.710338],accel_mss,speed_ms,0,blend_radius_m)
    |   movel([0.139542, -1.267692, -2.622419, -0.822278, 1.570796, 1.710338],accel_mss,speed_ms,0,blend_radius_m)
    |   movel([0.136902, -1.272677, -2.619596, -0.820115, 1.570796, 1.707698],accel_mss,speed_ms,0,blend_radius_m)
    |   movel([0.136902, -1.295634, -2.630639, -0.786116, 1.570796, 1.707698],accel_mss,speed_ms,0,blend_radius_m)
    |   movel([0.138776, -1.295655, -2.630626, -0.786107, 1.570796, 1.709572],accel_mss,speed_ms,0,blend_radius_m)
    |   movel([0.139217, -1.296896, -2.629895, -0.785597, 1.570796, 1.710014],accel_mss,speed_ms,0,blend_radius_m)
    |   movel([0.138293, -1.298605, -2.628885, -0.784899, 1.570796, 1.709090],accel_mss,speed_ms,0,blend_radius_m)
    |   movel([0.136589, -1.299673, -2.628252, -0.784464, 1.570796, 1.707385],accel_mss,speed_ms,0,blend_radius_m)
    |   movel([0.109164, -1.307965, -2.623286, -0.781138, 1.570796, 1.679961],accel_mss,speed_ms,0,blend_radius_m)
    |   movel([0.107634, -1.307884, -2.623335, -0.781170, 1.570796, 1.678430],accel_mss,speed_ms,0,blend_radius_m)
    |   movel([0.107124, -1.306654, -2.624077, -0.781658, 1.570796, 1.677920],accel_mss,speed_ms,0,blend_radius_m)
    |   movel([0.107957, -1.305023, -2.625058, -0.782308, 1.570796, 1.678753],accel_mss,speed_ms,0,blend_radius_m)
    |   movel([0.109665, -1.303923, -2.625718, -0.782748, 1.570796, 1.680461],accel_mss,speed_ms,0,blend_radius_m)
    |   movel([0.136902, -1.295634, -2.630639, -0.786116, 1.570796, 1.707698],accel_mss,speed_ms,0,blend_radius_m)
    |   movel([0.138776, -1.295655, -2.630626, -0.786107, 1.570796, 1.709572],accel_mss,speed_ms,0,blend_radius_m)
    |   movel([0.139217, -1.296896, -2.629895, -0.785597, 1.570796, 1.710014],accel_mss,speed_ms,0,blend_radius_m)
    |   movel([0.138293, -1.298605, -2.628885, -0.784899, 1.570796, 1.709090],accel_mss,speed_ms,0,blend_radius_m)
    |   movel([0.136589, -1.299673, -2.628252, -0.784464, 1.570796, 1.707385],accel_mss,speed_ms,0,blend_radius_m)
    |   movel([0.109164, -1.307965, -2.623286, -0.781138, 1.570796, 1.679961],accel_mss,speed_ms,0,blend_radius_m)
    |   movel([0.107634, -1.307884, -2.623335, -0.781170, 1.570796, 1.678430],accel_mss,speed_ms,0,blend_radius_m)
    |   movel([0.107124, -1.306654, -2.624077, -0.781658, 1.570796, 1.677920],accel_mss,speed_ms,0,blend_radius_m)
    |   movel([0.107957, -1.305023, -2.625058, -0.782308, 1.570796, 1.678753],accel_mss,speed_ms,0,blend_radius_m)
    |   movel([0.109665, -1.303923, -2.625718, -0.782748, 1.570796, 1.680461],accel_mss,speed_ms,0,blend_radius_m)
    |   movel([0.136902, -1.295634, -2.630639, -0.786116, 1.570796, 1.707698],accel_mss,speed_ms,0,blend_radius_m)
    |   movel([0.136902, -1.272677, -2.619596, -0.820115, 1.570796, 1.707698],accel_mss,speed_ms,0,blend_radius_m)
    |   movel([0.102588, -1.292594, -2.608012, -0.811784, 1.570796, 1.673385],accel_mss,speed_ms,0,blend_radius_m)
    |   movel([0.102588, -1.315277, -2.618832, -0.778280, 1.570796, 1.673385],accel_mss,speed_ms,0,blend_radius_m)
    |   movel([0.102118, -1.319312, -2.616344, -0.776734, 1.570796, 1.672914],accel_mss,speed_ms,0,blend_radius_m)
    |   movel([0.103716, -1.319458, -2.616253, -0.776678, 1.570796, 1.674512],accel_mss,speed_ms,0,blend_radius_m)
    |   movel([0.104787, -1.320410, -2.615663, -0.776316, 1.570796, 1.675583],accel_mss,speed_ms,0,blend_radius_m)
    |   movel([0.105005, -1.321842, -2.614772, -0.775775, 1.570796, 1.675802],accel_mss,speed_ms,0,blend_radius_m)
    |   movel([0.104498, -1.323379, -2.613813, -0.775196, 1.570796, 1.675294],accel_mss,speed_ms,0,blend_radius_m)
    |   movel([0.103009, -1.325238, -2.612650, -0.774501, 1.570796, 1.673805],accel_mss,speed_ms,0,blend_radius_m)
    |   movel([0.101298, -1.326378, -2.611934, -0.774077, 1.570796, 1.672094],accel_mss,speed_ms,0,blend_radius_m)
    |   movel([0.100827, -1.330449, -2.609362, -0.772577, 1.570796, 1.671623],accel_mss,speed_ms,0,blend_radius_m)
    |   movel([0.099266, -1.330928, -2.609058, -0.772402, 1.570796, 1.670062],accel_mss,speed_ms,0,blend_radius_m)
    |   movel([0.099729, -1.326862, -2.611629, -0.773898, 1.570796, 1.670526],accel_mss,speed_ms,0,blend_radius_m)
    |   movel([0.098466, -1.326822, -2.611654, -0.773913, 1.570796, 1.669263],accel_mss,speed_ms,0,blend_radius_m)
    |   movel([0.097449, -1.326310, -2.611976, -0.774103, 1.570796, 1.668246],accel_mss,speed_ms,0,blend_radius_m)
    |   movel([0.096901, -1.325414, -2.612540, -0.774436, 1.570796, 1.667698],accel_mss,speed_ms,0,blend_radius_m)
    |   movel([0.096821, -1.324381, -2.613187, -0.774821, 1.570796, 1.667618],accel_mss,speed_ms,0,blend_radius_m)
    |   movel([0.097620, -1.322342, -2.614461, -0.775586, 1.570796, 1.668416],accel_mss,speed_ms,0,blend_radius_m)
    |   movel([0.098713, -1.321062, -2.615257, -0.776069, 1.570796, 1.669510],accel_mss,speed_ms,0,blend_radius_m)
    |   movel([0.099700, -1.320284, -2.615741, -0.776364, 1.570796, 1.670496],accel_mss,speed_ms,0,blend_radius_m)
    |   movel([0.100536, -1.319805, -2.616038, -0.776546, 1.570796, 1.671333],accel_mss,speed_ms,0,blend_radius_m)
    |   movel([0.100999, -1.315775, -2.618526, -0.778088, 1.570796, 1.671796],accel_mss,speed_ms,0,blend_radius_m)
    |   movel([0.102588, -1.315277, -2.618832, -0.778280, 1.570796, 1.673385],accel_mss,speed_ms,0,blend_radius_m)
    |   movel([0.102118, -1.319312, -2.616344, -0.776734, 1.570796, 1.672914],accel_mss,speed_ms,0,blend_radius_m)
    |   movel([0.103716, -1.319458, -2.616253, -0.776678, 1.570796, 1.674512],accel_mss,speed_ms,0,blend_radius_m)
    |   movel([0.104787, -1.320410, -2.615663, -0.776316, 1.570796, 1.675583],accel_mss,speed_ms,0,blend_radius_m)
    |   movel([0.105005, -1.321842, -2.614772, -0.775775, 1.570796, 1.675802],accel_mss,speed_ms,0,blend_radius_m)
    |   movel([0.104498, -1.323379, -2.613813, -0.775196, 1.570796, 1.675294],accel_mss,speed_ms,0,blend_radius_m)
    |   movel([0.103009, -1.325238, -2.612650, -0.774501, 1.570796, 1.673805],accel_mss,speed_ms,0,blend_radius_m)
    |   movel([0.101298, -1.326378, -2.611934, -0.774077, 1.570796, 1.672094],accel_mss,speed_ms,0,blend_radius_m)
    |   movel([0.100827, -1.330449, -2.609362, -0.772577, 1.570796, 1.671623],accel_mss,speed_ms,0,blend_radius_m)
    |   movel([0.099266, -1.330928, -2.609058, -0.772402, 1.570796, 1.670062],accel_mss,speed_ms,0,blend_radius_m)
    |   movel([0.099729, -1.326862, -2.611629, -0.773898, 1.570796, 1.670526],accel_mss,speed_ms,0,blend_radius_m)
    |   movel([0.098466, -1.326822, -2.611654, -0.773913, 1.570796, 1.669263],accel_mss,speed_ms,0,blend_radius_m)
    |   movel([0.097449, -1.326310, -2.611976, -0.774103, 1.570796, 1.668246],accel_mss,speed_ms,0,blend_radius_m)
    |   movel([0.096901, -1.325414, -2.612540, -0.774436, 1.570796, 1.667698],accel_mss,speed_ms,0,blend_radius_m)
    |   movel([0.096821, -1.324381, -2.613187, -0.774821, 1.570796, 1.667618],accel_mss,speed_ms,0,blend_radius_m)
    |   movel([0.097620, -1.322342, -2.614461, -0.775586, 1.570796, 1.668416],accel_mss,speed_ms,0,blend_radius_m)
    |   movel([0.098713, -1.321062, -2.615257, -0.776069, 1.570796, 1.669510],accel_mss,speed_ms,0,blend_radius_m)
    |   movel([0.099700, -1.320284, -2.615741, -0.776364, 1.570796, 1.670496],accel_mss,speed_ms,0,blend_radius_m)
    |   movel([0.100536, -1.319805, -2.616038, -0.776546, 1.570796, 1.671333],accel_mss,speed_ms,0,blend_radius_m)
    |   movel([0.100999, -1.315775, -2.618526, -0.778088, 1.570796, 1.671796],accel_mss,speed_ms,0,blend_radius_m)
    |   movel([0.102588, -1.315277, -2.618832, -0.778280, 1.570796, 1.673385],accel_mss,speed_ms,0,blend_radius_m)
    |   movel([0.102588, -1.292594, -2.608012, -0.811784, 1.570796, 1.673385],accel_mss,speed_ms,0,blend_radius_m)
    |   movel([0.110621, -1.295684, -2.606170, -0.810535, 1.570796, 1.681418],accel_mss,speed_ms,0,blend_radius_m)
    |   movel([0.110621, -1.318323, -2.616955, -0.777111, 1.570796, 1.681418],accel_mss,speed_ms,0,blend_radius_m)
    |   movel([0.111733, -1.317041, -2.617747, -0.777602, 1.570796, 1.682529],accel_mss,speed_ms,0,blend_radius_m)
    |   movel([0.112731, -1.316265, -2.618225, -0.777900, 1.570796, 1.683527],accel_mss,speed_ms,0,blend_radius_m)
    |   movel([0.113573, -1.315789, -2.618517, -0.778083, 1.570796, 1.684370],accel_mss,speed_ms,0,blend_radius_m)
    |   movel([0.114098, -1.311716, -2.621010, -0.779663, 1.570796, 1.684895],accel_mss,speed_ms,0,blend_radius_m)
    |   movel([0.115693, -1.311230, -2.621306, -0.779853, 1.570796, 1.686489],accel_mss,speed_ms,0,blend_radius_m)
    |   movel([0.115160, -1.315308, -2.618812, -0.778268, 1.570796, 1.685956],accel_mss,speed_ms,0,blend_radius_m)
    |   movel([0.116767, -1.315470, -2.618713, -0.778206, 1.570796, 1.687563],accel_mss,speed_ms,0,blend_radius_m)
    |   movel([0.117821, -1.316447, -2.618113, -0.777830, 1.570796, 1.688618],accel_mss,speed_ms,0,blend_radius_m)
    |   movel([0.118017, -1.317898, -2.617218, -0.777273, 1.570796, 1.688814],accel_mss,speed_ms,0,blend_radius_m)
    |   movel([0.117473, -1.319452, -2.616257, -0.776680, 1.570796, 1.688269],accel_mss,speed_ms,0,blend_radius_m)
    |   movel([0.115957, -1.321315, -2.615100, -0.775974, 1.570796, 1.686753],accel_mss,speed_ms,0,blend_radius_m)
    |   movel([0.114231, -1.322449, -2.614394, -0.775546, 1.570796, 1.685027],accel_mss,speed_ms,0,blend_radius_m)
    |   movel([0.113698, -1.326563, -2.611817, -0.774009, 1.570796, 1.684494],accel_mss,speed_ms,0,blend_radius_m)
    |   movel([0.112132, -1.327030, -2.611524, -0.773836, 1.570796, 1.682928],accel_mss,speed_ms,0,blend_radius_m)
    |   movel([0.112657, -1.322921, -2.614100, -0.775369, 1.570796, 1.683454],accel_mss,speed_ms,0,blend_radius_m)
    |   movel([0.111397, -1.322866, -2.614134, -0.775389, 1.570796, 1.682193],accel_mss,speed_ms,0,blend_radius_m)
    |   movel([0.110403, -1.322332, -2.614467, -0.775590, 1.570796, 1.681199],accel_mss,speed_ms,0,blend_radius_m)
    |   movel([0.109856, -1.321423, -2.615033, -0.775933, 1.570796, 1.680653],accel_mss,speed_ms,0,blend_radius_m)
    |   movel([0.109806, -1.320373, -2.615685, -0.776330, 1.570796, 1.680602],accel_mss,speed_ms,0,blend_radius_m)
    |   movel([0.110621, -1.318323, -2.616955, -0.777111, 1.570796, 1.681418],accel_mss,speed_ms,0,blend_radius_m)
    |   movel([0.111733, -1.317041, -2.617747, -0.777602, 1.570796, 1.682529],accel_mss,speed_ms,0,blend_radius_m)
    |   movel([0.112731, -1.316265, -2.618225, -0.777900, 1.570796, 1.683527],accel_mss,speed_ms,0,blend_radius_m)
    |   movel([0.113573, -1.315789, -2.618517, -0.778083, 1.570796, 1.684370],accel_mss,speed_ms,0,blend_radius_m)
    |   movel([0.114098, -1.311716, -2.621010, -0.779663, 1.570796, 1.684895],accel_mss,speed_ms,0,blend_radius_m)
    |   movel([0.115693, -1.311230, -2.621306, -0.779853, 1.570796, 1.686489],accel_mss,speed_ms,0,blend_radius_m)
    |   movel([0.115160, -1.315308, -2.618812, -0.778268, 1.570796, 1.685956],accel_mss,speed_ms,0,blend_radius_m)
    |   movel([0.116767, -1.315470, -2.618713, -0.778206, 1.570796, 1.687563],accel_mss,speed_ms,0,blend_radius_m)
    |   movel([0.117821, -1.316447, -2.618113, -0.777830, 1.570796, 1.688618],accel_mss,speed_ms,0,blend_radius_m)
    |   movel([0.118017, -1.317898, -2.617218, -0.777273, 1.570796, 1.688814],accel_mss,speed_ms,0,blend_radius_m)
    |   movel([0.117473, -1.319452, -2.616257, -0.776680, 1.570796, 1.688269],accel_mss,speed_ms,0,blend_radius_m)
    |   movel([0.115957, -1.321315, -2.615100, -0.775974, 1.570796, 1.686753],accel_mss,speed_ms,0,blend_radius_m)
    |   movel([0.114231, -1.322449, -2.614394, -0.775546, 1.570796, 1.685027],accel_mss,speed_ms,0,blend_radius_m)
    |   movel([0.113698, -1.326563, -2.611817, -0.774009, 1.570796, 1.684494],accel_mss,speed_ms,0,blend_radius_m)
    |   movel([0.112132, -1.327030, -2.611524, -0.773836, 1.570796, 1.682928],accel_mss,speed_ms,0,blend_radius_m)
    |   movel([0.112657, -1.322921, -2.614100, -0.775369, 1.570796, 1.683454],accel_mss,speed_ms,0,blend_radius_m)
    |   movel([0.111397, -1.322866, -2.614134, -0.775389, 1.570796, 1.682193],accel_mss,speed_ms,0,blend_radius_m)
    |   movel([0.110403, -1.322332, -2.614467, -0.775590, 1.570796, 1.681199],accel_mss,speed_ms,0,blend_radius_m)
    |   movel([0.109856, -1.321423, -2.615033, -0.775933, 1.570796, 1.680653],accel_mss,speed_ms,0,blend_radius_m)
    |   movel([0.109806, -1.320373, -2.615685, -0.776330, 1.570796, 1.680602],accel_mss,speed_ms,0,blend_radius_m)
    |   movel([0.110621, -1.318323, -2.616955, -0.777111, 1.570796, 1.681418],accel_mss,speed_ms,0,blend_radius_m)
    |   movel([0.110621, -1.295684, -2.606170, -0.810535, 1.570796, 1.681418],accel_mss,speed_ms,0,blend_radius_m)
    |   movel([0.124027, -1.293327, -2.607575, -0.811486, 1.570796, 1.694824],accel_mss,speed_ms,0,blend_radius_m)
    |   movel([0.124027, -1.316000, -2.618388, -0.778001, 1.570796, 1.694824],accel_mss,speed_ms,0,blend_radius_m)
    |   movel([0.124875, -1.313945, -2.619648, -0.778796, 1.570796, 1.695671],accel_mss,speed_ms,0,blend_radius_m)
    |   movel([0.126008, -1.312648, -2.620441, -0.779300, 1.570796, 1.696805],accel_mss,speed_ms,0,blend_radius_m)
    |   movel([0.127031, -1.311870, -2.620916, -0.779603, 1.570796, 1.697827],accel_mss,speed_ms,0,blend_radius_m)
    |   movel([0.127879, -1.311412, -2.621195, -0.779782, 1.570796, 1.698675],accel_mss,speed_ms,0,blend_radius_m)
    |   movel([0.128473, -1.307291, -2.623693, -0.781405, 1.570796, 1.699269],accel_mss,speed_ms,0,blend_radius_m)
    |   movel([0.130059, -1.306823, -2.623975, -0.781591, 1.570796, 1.700856],accel_mss,speed_ms,0,blend_radius_m)
    |   movel([0.129457, -1.310949, -2.621477, -0.779963, 1.570796, 1.700254],accel_mss,speed_ms,0,blend_radius_m)
    |   movel([0.131059, -1.311133, -2.621365, -0.779891, 1.570796, 1.701855],accel_mss,speed_ms,0,blend_radius_m)
    |   movel([0.132096, -1.312124, -2.620761, -0.779504, 1.570796, 1.702893],accel_mss,speed_ms,0,blend_radius_m)
    |   movel([0.132267, -1.313596, -2.619862, -0.778931, 1.570796, 1.703063],accel_mss,speed_ms,0,blend_radius_m)
    |   movel([0.131711, -1.315160, -2.618904, -0.778326, 1.570796, 1.702507],accel_mss,speed_ms,0,blend_radius_m)
    |   movel([0.130151, -1.317044, -2.617745, -0.777600, 1.570796, 1.700947],accel_mss,speed_ms,0,blend_radius_m)
    |   movel([0.128408, -1.318170, -2.617050, -0.777169, 1.570796, 1.699205],accel_mss,speed_ms,0,blend_radius_m)
    |   movel([0.127806, -1.322331, -2.614468, -0.775591, 1.570796, 1.698603],accel_mss,speed_ms,0,blend_radius_m)
    |   movel([0.126249, -1.322780, -2.614188, -0.775422, 1.570796, 1.697045],accel_mss,speed_ms,0,blend_radius_m)
    |   movel([0.126843, -1.318625, -2.616769, -0.776995, 1.570796, 1.697639],accel_mss,speed_ms,0,blend_radius_m)
    |   movel([0.125585, -1.318553, -2.616813, -0.777023, 1.570796, 1.696382],accel_mss,speed_ms,0,blend_radius_m)
    |   movel([0.124589, -1.318004, -2.617152, -0.777232, 1.570796, 1.695385],accel_mss,speed_ms,0,blend_radius_m)
    |   movel([0.124073, -1.317060, -2.617735, -0.777594, 1.570796, 1.694870],accel_mss,speed_ms,0,blend_radius_m)
    |   movel([0.124027, -1.316000, -2.618388, -0.778001, 1.570796, 1.694824],accel_mss,speed_ms,0,blend_radius_m)
    |   movel([0.124875, -1.313945, -2.619648, -0.778796, 1.570796, 1.695671],accel_mss,speed_ms,0,blend_radius_m)
    |   movel([0.126008, -1.312648, -2.620441, -0.779300, 1.570796, 1.696805],accel_mss,speed_ms,0,blend_radius_m)
    |   movel([0.127031, -1.311870, -2.620916, -0.779603, 1.570796, 1.697827],accel_mss,speed_ms,0,blend_radius_m)
    |   movel([0.127879, -1.311412, -2.621195, -0.779782, 1.570796, 1.698675],accel_mss,speed_ms,0,blend_radius_m)
    |   movel([0.128473, -1.307291, -2.623693, -0.781405, 1.570796, 1.699269],accel_mss,speed_ms,0,blend_radius_m)
    |   movel([0.130059, -1.306823, -2.623975, -0.781591, 1.570796, 1.700856],accel_mss,speed_ms,0,blend_radius_m)
    |   movel([0.129457, -1.310949, -2.621477, -0.779963, 1.570796, 1.700254],accel_mss,speed_ms,0,blend_radius_m)
    |   movel([0.131059, -1.311133, -2.621365, -0.779891, 1.570796, 1.701855],accel_mss,speed_ms,0,blend_radius_m)
    |   movel([0.132096, -1.312124, -2.620761, -0.779504, 1.570796, 1.702893],accel_mss,speed_ms,0,blend_radius_m)
    |   movel([0.132267, -1.313596, -2.619862, -0.778931, 1.570796, 1.703063],accel_mss,speed_ms,0,blend_radius_m)
    |   movel([0.131711, -1.315160, -2.618904, -0.778326, 1.570796, 1.702507],accel_mss,speed_ms,0,blend_radius_m)
    |   movel([0.130151, -1.317044, -2.617745, -0.777600, 1.570796, 1.700947],accel_mss,speed_ms,0,blend_radius_m)
    |   movel([0.128408, -1.318170, -2.617050, -0.777169, 1.570796, 1.699205],accel_mss,speed_ms,0,blend_radius_m)
    |   movel([0.127806, -1.322331, -2.614468, -0.775591, 1.570796, 1.698603],accel_mss,speed_ms,0,blend_radius_m)
    |   movel([0.126249, -1.322780, -2.614188, -0.775422, 1.570796, 1.697045],accel_mss,speed_ms,0,blend_radius_m)
    |   movel([0.126843, -1.318625, -2.616769, -0.776995, 1.570796, 1.697639],accel_mss,speed_ms,0,blend_radius_m)
    |   movel([0.125585, -1.318553, -2.616813, -0.777023, 1.570796, 1.696382],accel_mss,speed_ms,0,blend_radius_m)
    |   movel([0.124589, -1.318004, -2.617152, -0.777232, 1.570796, 1.695385],accel_mss,speed_ms,0,blend_radius_m)
    |   movel([0.124073, -1.317060, -2.617735, -0.777594, 1.570796, 1.694870],accel_mss,speed_ms,0,blend_radius_m)
    |   movel([0.124027, -1.316000, -2.618388, -0.778001, 1.570796, 1.694824],accel_mss,speed_ms,0,blend_radius_m)
    |   movel([0.124027, -1.293327, -2.607575, -0.811486, 1.570796, 1.694824],accel_mss,speed_ms,0,blend_radius_m)
    |   movel([0.139312, -1.304021, -2.601139, -0.807229, 1.570796, 1.710108],accel_mss,speed_ms,0,blend_radius_m)
    |   movel([0.139312, -1.326538, -2.611833, -0.774018, 1.570796, 1.710108],accel_mss,speed_ms,0,blend_radius_m)
    |   movel([0.137968, -1.327548, -2.611197, -0.773644, 1.570796, 1.708764],accel_mss,speed_ms,0,blend_radius_m)
    |   movel([0.137454, -1.328804, -2.610404, -0.773181, 1.570796, 1.708250],accel_mss,speed_ms,0,blend_radius_m)
    |   movel([0.138010, -1.329729, -2.609819, -0.772841, 1.570796, 1.708806],accel_mss,speed_ms,0,blend_radius_m)
    |   movel([0.139318, -1.329665, -2.609860, -0.772865, 1.570796, 1.710114],accel_mss,speed_ms,0,blend_radius_m)
    |   movel([0.157503, -1.322871, -2.614131, -0.775387, 1.570796, 1.728299],accel_mss,speed_ms,0,blend_radius_m)
    |   movel([0.158808, -1.321908, -2.614731, -0.775750, 1.570796, 1.729604],accel_mss,speed_ms,0,blend_radius_m)
    |   movel([0.159327, -1.320712, -2.615475, -0.776202, 1.570796, 1.730123],accel_mss,speed_ms,0,blend_radius_m)
    |   movel([0.158776, -1.319783, -2.616052, -0.776554, 1.570796, 1.729572],accel_mss,speed_ms,0,blend_radius_m)
    |   movel([0.157605, -1.319826, -2.616025, -0.776538, 1.570796, 1.728401],accel_mss,speed_ms,0,blend_radius_m)
    |   movel([0.139407, -1.326501, -2.611857, -0.774032, 1.570796, 1.710204],accel_mss,speed_ms,0,blend_radius_m)
    |   movel([0.157605, -1.319826, -2.616025, -0.776538, 1.570796, 1.728401],accel_mss,speed_ms,0,blend_radius_m)
    |   movel([0.158776, -1.319783, -2.616052, -0.776554, 1.570796, 1.729572],accel_mss,speed_ms,0,blend_radius_m)
    |   movel([0.159327, -1.320712, -2.615475, -0.776202, 1.570796, 1.730123],accel_mss,speed_ms,0,blend_radius_m)
    |   movel([0.158808, -1.321908, -2.614731, -0.775750, 1.570796, 1.729604],accel_mss,speed_ms,0,blend_radius_m)
    |   movel([0.157503, -1.322871, -2.614131, -0.775387, 1.570796, 1.728299],accel_mss,speed_ms,0,blend_radius_m)
    |   movel([0.139318, -1.329665, -2.609860, -0.772865, 1.570796, 1.710114],accel_mss,speed_ms,0,blend_radius_m)
    |   movel([0.138010, -1.329729, -2.609819, -0.772841, 1.570796, 1.708806],accel_mss,speed_ms,0,blend_radius_m)
    |   movel([0.137454, -1.328804, -2.610404, -0.773181, 1.570796, 1.708250],accel_mss,speed_ms,0,blend_radius_m)
    |   movel([0.137968, -1.327548, -2.611197, -0.773644, 1.570796, 1.708764],accel_mss,speed_ms,0,blend_radius_m)
    |   movel([0.139312, -1.326538, -2.611833, -0.774018, 1.570796, 1.710108],accel_mss,speed_ms,0,blend_radius_m)
    |   movel([0.139312, -1.304021, -2.601139, -0.807229, 1.570796, 1.710108],accel_mss,speed_ms,0,blend_radius_m)
    |   movel([0.137121, -1.308497, -2.598402, -0.805490, 1.570796, 1.707917],accel_mss,speed_ms,0,blend_radius_m)
    |   movel([0.137121, -1.330949, -2.609046, -0.772395, 1.570796, 1.707917],accel_mss,speed_ms,0,blend_radius_m)
    |   movel([0.159178, -1.322478, -2.614376, -0.775535, 1.570796, 1.729975],accel_mss,speed_ms,0,blend_radius_m)
    |   movel([0.158191, -1.326748, -2.611701, -0.773940, 1.570796, 1.728988],accel_mss,speed_ms,0,blend_radius_m)
    |   movel([0.156099, -1.328980, -2.610293, -0.773116, 1.570796, 1.726896],accel_mss,speed_ms,0,blend_radius_m)
    |   movel([0.152278, -1.332271, -2.608204, -0.771913, 1.570796, 1.723074],accel_mss,speed_ms,0,blend_radius_m)
    |   movel([0.145547, -1.336291, -2.605634, -0.770464, 1.570796, 1.716343],accel_mss,speed_ms,0,blend_radius_m)
    |   movel([0.141868, -1.337687, -2.604736, -0.769966, 1.570796, 1.712664],accel_mss,speed_ms,0,blend_radius_m)
    |   movel([0.138205, -1.338537, -2.604188, -0.769664, 1.570796, 1.709002],accel_mss,speed_ms,0,blend_radius_m)
    |   movel([0.135914, -1.338766, -2.604040, -0.769583, 1.570796, 1.706710],accel_mss,speed_ms,0,blend_radius_m)
    |   movel([0.137121, -1.330949, -2.609046, -0.772395, 1.570796, 1.707917],accel_mss,speed_ms,0,blend_radius_m)
    |   movel([0.159178, -1.322478, -2.614376, -0.775535, 1.570796, 1.729975],accel_mss,speed_ms,0,blend_radius_m)
    |   movel([0.158191, -1.326748, -2.611701, -0.773940, 1.570796, 1.728988],accel_mss,speed_ms,0,blend_radius_m)
    |   movel([0.156099, -1.328980, -2.610293, -0.773116, 1.570796, 1.726896],accel_mss,speed_ms,0,blend_radius_m)
    |   movel([0.152278, -1.332271, -2.608204, -0.771913, 1.570796, 1.723074],accel_mss,speed_ms,0,blend_radius_m)
    |   movel([0.145547, -1.336291, -2.605634, -0.770464, 1.570796, 1.716343],accel_mss,speed_ms,0,blend_radius_m)
    |   movel([0.141868, -1.337687, -2.604736, -0.769966, 1.570796, 1.712664],accel_mss,speed_ms,0,blend_radius_m)
    |   movel([0.138205, -1.338537, -2.604188, -0.769664, 1.570796, 1.709002],accel_mss,speed_ms,0,blend_radius_m)
    |   movel([0.135914, -1.338766, -2.604040, -0.769583, 1.570796, 1.706710],accel_mss,speed_ms,0,blend_radius_m)
    |   movel([0.137121, -1.330949, -2.609046, -0.772395, 1.570796, 1.707917],accel_mss,speed_ms,0,blend_radius_m)
    |   movel([0.137121, -1.308497, -2.598402, -0.805490, 1.570796, 1.707917],accel_mss,speed_ms,0,blend_radius_m)
    |   movel([0.139265, -1.307209, -2.599192, -0.805988, 1.570796, 1.710061],accel_mss,speed_ms,0,blend_radius_m)
    |   movel([0.139265, -1.329680, -2.609850, -0.772859, 1.570796, 1.710061],accel_mss,speed_ms,0,blend_radius_m)
    |   movel([0.157503, -1.322871, -2.614131, -0.775387, 1.570796, 1.728299],accel_mss,speed_ms,0,blend_radius_m)
    |   movel([0.139265, -1.329680, -2.609850, -0.772859, 1.570796, 1.710061],accel_mss,speed_ms,0,blend_radius_m)
    |   movel([0.139265, -1.307209, -2.599192, -0.805988, 1.570796, 1.710061],accel_mss,speed_ms,0,blend_radius_m)
    |   movel([0.157605, -1.297209, -2.605256, -0.809924, 1.570796, 1.728401],accel_mss,speed_ms,0,blend_radius_m)
    |   movel([0.157605, -1.319826, -2.616025, -0.776538, 1.570796, 1.728401],accel_mss,speed_ms,0,blend_radius_m)
    |   movel([0.139325, -1.326535, -2.611835, -0.774019, 1.570796, 1.710122],accel_mss,speed_ms,0,blend_radius_m)
    |   movel([0.157605, -1.319826, -2.616025, -0.776538, 1.570796, 1.728401],accel_mss,speed_ms,0,blend_radius_m)
    |   movel([0.157605, -1.297209, -2.605256, -0.809924, 1.570796, 1.728401],accel_mss,speed_ms,0,blend_radius_m)
    |   movel([0.128953, -1.337126, -2.580273, -0.794990, 1.570796, 1.699749],accel_mss,speed_ms,0,blend_radius_m)
    |   movel([0.128953, -1.359134, -2.590602, -0.762653, 1.570796, 1.699749],accel_mss,speed_ms,0,blend_radius_m)
    |   movel([0.129931, -1.359112, -2.590617, -0.762660, 1.570796, 1.700727],accel_mss,speed_ms,0,blend_radius_m)
    |   movel([0.130637, -1.360335, -2.589792, -0.762262, 1.570796, 1.701433],accel_mss,speed_ms,0,blend_radius_m)
    |   movel([0.128801, -1.372693, -2.581334, -0.758361, 1.570796, 1.699597],accel_mss,speed_ms,0,blend_radius_m)
    |   movel([0.128085, -1.374008, -2.580422, -0.757959, 1.570796, 1.698881],accel_mss,speed_ms,0,blend_radius_m)
    |   movel([0.126649, -1.374860, -2.579829, -0.757700, 1.570796, 1.697446],accel_mss,speed_ms,0,blend_radius_m)
    |   movel([0.125549, -1.374830, -2.579850, -0.757709, 1.570796, 1.696346],accel_mss,speed_ms,0,blend_radius_m)
    |   movel([0.124984, -1.373693, -2.580641, -0.758055, 1.570796, 1.695780],accel_mss,speed_ms,0,blend_radius_m)
    |   movel([0.126764, -1.361368, -2.589093, -0.761928, 1.570796, 1.697560],accel_mss,speed_ms,0,blend_radius_m)
    |   movel([0.127648, -1.359863, -2.590111, -0.762415, 1.570796, 1.698445],accel_mss,speed_ms,0,blend_radius_m)
    |   movel([0.128953, -1.359134, -2.590602, -0.762653, 1.570796, 1.699749],accel_mss,speed_ms,0,blend_radius_m)
    |   movel([0.129931, -1.359112, -2.590617, -0.762660, 1.570796, 1.700727],accel_mss,speed_ms,0,blend_radius_m)
    |   movel([0.130637, -1.360335, -2.589792, -0.762262, 1.570796, 1.701433],accel_mss,speed_ms,0,blend_radius_m)
    |   movel([0.128801, -1.372693, -2.581334, -0.758361, 1.570796, 1.699597],accel_mss,speed_ms,0,blend_radius_m)
    |   movel([0.128085, -1.374008, -2.580422, -0.757959, 1.570796, 1.698881],accel_mss,speed_ms,0,blend_radius_m)
    |   movel([0.126649, -1.374860, -2.579829, -0.757700, 1.570796, 1.697446],accel_mss,speed_ms,0,blend_radius_m)
    |   movel([0.125549, -1.374830, -2.579850, -0.757709, 1.570796, 1.696346],accel_mss,speed_ms,0,blend_radius_m)
    |   movel([0.124984, -1.373693, -2.580641, -0.758055, 1.570796, 1.695780],accel_mss,speed_ms,0,blend_radius_m)
    |   movel([0.126764, -1.361368, -2.589093, -0.761928, 1.570796, 1.697560],accel_mss,speed_ms,0,blend_radius_m)
    |   movel([0.127648, -1.359863, -2.590111, -0.762415, 1.570796, 1.698445],accel_mss,speed_ms,0,blend_radius_m)
    |   movel([0.128953, -1.359134, -2.590602, -0.762653, 1.570796, 1.699749],accel_mss,speed_ms,0,blend_radius_m)
    |   movel([0.128953, -1.337126, -2.580273, -0.794990, 1.570796, 1.699749],accel_mss,speed_ms,0,blend_radius_m)
    |   movel([0.115112, -1.350051, -2.571731, -0.790607, 1.570796, 1.685908],accel_mss,speed_ms,0,blend_radius_m)
    |   movel([0.115112, -1.371849, -2.581919, -0.758621, 1.570796, 1.685908],accel_mss,speed_ms,0,blend_radius_m)
    |   movel([0.116193, -1.373352, -2.580877, -0.758160, 1.570796, 1.686989],accel_mss,speed_ms,0,blend_radius_m)
    |   movel([0.116249, -1.374664, -2.579965, -0.757760, 1.570796, 1.687045],accel_mss,speed_ms,0,blend_radius_m)
    |   movel([0.115874, -1.376005, -2.579031, -0.757353, 1.570796, 1.686671],accel_mss,speed_ms,0,blend_radius_m)
    |   movel([0.114185, -1.378394, -2.577359, -0.756635, 1.570796, 1.684981],accel_mss,speed_ms,0,blend_radius_m)
    |   movel([0.112473, -1.379710, -2.576435, -0.756244, 1.570796, 1.683269],accel_mss,speed_ms,0,blend_radius_m)
    |   movel([0.110585, -1.380538, -2.575852, -0.755998, 1.570796, 1.681381],accel_mss,speed_ms,0,blend_radius_m)
    |   movel([0.107531, -1.380532, -2.575857, -0.756000, 1.570796, 1.678328],accel_mss,speed_ms,0,blend_radius_m)
    |   movel([0.106059, -1.379087, -2.576873, -0.756429, 1.570796, 1.676856],accel_mss,speed_ms,0,blend_radius_m)
    |   movel([0.105889, -1.377500, -2.577986, -0.756903, 1.570796, 1.676686],accel_mss,speed_ms,0,blend_radius_m)
    |   movel([0.106393, -1.375882, -2.579117, -0.757390, 1.570796, 1.677189],accel_mss,speed_ms,0,blend_radius_m)
    |   movel([0.107428, -1.374324, -2.580202, -0.757863, 1.570796, 1.678224],accel_mss,speed_ms,0,blend_radius_m)
    |   movel([0.109711, -1.372396, -2.581540, -0.758453, 1.570796, 1.680507],accel_mss,speed_ms,0,blend_radius_m)
    |   movel([0.111551, -1.371590, -2.582098, -0.758701, 1.570796, 1.682347],accel_mss,speed_ms,0,blend_radius_m)
    |   movel([0.113864, -1.371391, -2.582236, -0.758762, 1.570796, 1.684661],accel_mss,speed_ms,0,blend_radius_m)
    |   movel([0.115112, -1.371849, -2.581919, -0.758621, 1.570796, 1.685908],accel_mss,speed_ms,0,blend_radius_m)
    |   movel([0.116193, -1.373352, -2.580877, -0.758160, 1.570796, 1.686989],accel_mss,speed_ms,0,blend_radius_m)
    |   movel([0.116249, -1.374664, -2.579965, -0.757760, 1.570796, 1.687045],accel_mss,speed_ms,0,blend_radius_m)
    |   movel([0.115874, -1.376005, -2.579031, -0.757353, 1.570796, 1.686671],accel_mss,speed_ms,0,blend_radius_m)
    |   movel([0.114185, -1.378394, -2.577359, -0.756635, 1.570796, 1.684981],accel_mss,speed_ms,0,blend_radius_m)
    |   movel([0.112473, -1.379710, -2.576435, -0.756244, 1.570796, 1.683269],accel_mss,speed_ms,0,blend_radius_m)
    |   movel([0.110585, -1.380538, -2.575852, -0.755998, 1.570796, 1.681381],accel_mss,speed_ms,0,blend_radius_m)
    |   movel([0.107531, -1.380532, -2.575857, -0.756000, 1.570796, 1.678328],accel_mss,speed_ms,0,blend_radius_m)
    |   movel([0.106059, -1.379087, -2.576873, -0.756429, 1.570796, 1.676856],accel_mss,speed_ms,0,blend_radius_m)
    |   movel([0.105889, -1.377500, -2.577986, -0.756903, 1.570796, 1.676686],accel_mss,speed_ms,0,blend_radius_m)
    |   movel([0.106393, -1.375882, -2.579117, -0.757390, 1.570796, 1.677189],accel_mss,speed_ms,0,blend_radius_m)
    |   movel([0.107428, -1.374324, -2.580202, -0.757863, 1.570796, 1.678224],accel_mss,speed_ms,0,blend_radius_m)
    |   movel([0.109711, -1.372396, -2.581540, -0.758453, 1.570796, 1.680507],accel_mss,speed_ms,0,blend_radius_m)
    |   movel([0.111551, -1.371590, -2.582098, -0.758701, 1.570796, 1.682347],accel_mss,speed_ms,0,blend_radius_m)
    |   movel([0.113864, -1.371391, -2.582236, -0.758762, 1.570796, 1.684661],accel_mss,speed_ms,0,blend_radius_m)
    |   movel([0.115112, -1.371849, -2.581919, -0.758621, 1.570796, 1.685908],accel_mss,speed_ms,0,blend_radius_m)
    |   movel([0.115112, -1.350051, -2.571731, -0.790607, 1.570796, 1.685908],accel_mss,speed_ms,0,blend_radius_m)
    |   movel([0.113017, -1.352274, -2.570239, -0.789876, 1.570796, 1.683814],accel_mss,speed_ms,0,blend_radius_m)
    |   movel([0.113017, -1.374036, -2.580403, -0.757951, 1.570796, 1.683814],accel_mss,speed_ms,0,blend_radius_m)
    |   movel([0.113544, -1.374762, -2.579898, -0.757730, 1.570796, 1.684340],accel_mss,speed_ms,0,blend_radius_m)
    |   movel([0.113571, -1.375390, -2.579460, -0.757539, 1.570796, 1.684368],accel_mss,speed_ms,0,blend_radius_m)
    |   movel([0.113388, -1.376043, -2.579004, -0.757342, 1.570796, 1.684185],accel_mss,speed_ms,0,blend_radius_m)
    |   movel([0.112582, -1.377193, -2.578201, -0.756995, 1.570796, 1.683378],accel_mss,speed_ms,0,blend_radius_m)
    |   movel([0.111746, -1.377832, -2.577753, -0.756804, 1.570796, 1.682542],accel_mss,speed_ms,0,blend_radius_m)
    |   movel([0.110831, -1.378240, -2.577468, -0.756682, 1.570796, 1.681627],accel_mss,speed_ms,0,blend_radius_m)
    |   movel([0.109362, -1.378230, -2.577474, -0.756684, 1.570796, 1.680158],accel_mss,speed_ms,0,blend_radius_m)
    |   movel([0.108648, -1.377530, -2.577965, -0.756894, 1.570796, 1.679444],accel_mss,speed_ms,0,blend_radius_m)
    |   movel([0.108562, -1.376761, -2.578503, -0.757125, 1.570796, 1.679358],accel_mss,speed_ms,0,blend_radius_m)
    |   movel([0.108807, -1.375975, -2.579052, -0.757362, 1.570796, 1.679603],accel_mss,speed_ms,0,blend_radius_m)
    |   movel([0.109317, -1.375221, -2.579578, -0.757590, 1.570796, 1.680113],accel_mss,speed_ms,0,blend_radius_m)
    |   movel([0.110409, -1.374305, -2.580215, -0.757869, 1.570796, 1.681205],accel_mss,speed_ms,0,blend_radius_m)
    |   movel([0.111301, -1.373912, -2.580489, -0.757989, 1.570796, 1.682097],accel_mss,speed_ms,0,blend_radius_m)
    |   movel([0.112411, -1.373819, -2.580553, -0.758017, 1.570796, 1.683208],accel_mss,speed_ms,0,blend_radius_m)
    |   movel([0.113017, -1.374036, -2.580403, -0.757951, 1.570796, 1.683814],accel_mss,speed_ms,0,blend_radius_m)
    |   movel([0.113544, -1.374762, -2.579898, -0.757730, 1.570796, 1.684340],accel_mss,speed_ms,0,blend_radius_m)
    |   movel([0.113571, -1.375390, -2.579460, -0.757539, 1.570796, 1.684368],accel_mss,speed_ms,0,blend_radius_m)
    |   movel([0.113388, -1.376043, -2.579004, -0.757342, 1.570796, 1.684185],accel_mss,speed_ms,0,blend_radius_m)
    |   movel([0.112582, -1.377193, -2.578201, -0.756995, 1.570796, 1.683378],accel_mss,speed_ms,0,blend_radius_m)
    |   movel([0.111746, -1.377832, -2.577753, -0.756804, 1.570796, 1.682542],accel_mss,speed_ms,0,blend_radius_m)
    |   movel([0.110831, -1.378240, -2.577468, -0.756682, 1.570796, 1.681627],accel_mss,speed_ms,0,blend_radius_m)
    |   movel([0.109362, -1.378230, -2.577474, -0.756684, 1.570796, 1.680158],accel_mss,speed_ms,0,blend_radius_m)
    |   movel([0.108648, -1.377530, -2.577965, -0.756894, 1.570796, 1.679444],accel_mss,speed_ms,0,blend_radius_m)
    |   movel([0.108562, -1.376761, -2.578503, -0.757125, 1.570796, 1.679358],accel_mss,speed_ms,0,blend_radius_m)
    |   movel([0.108807, -1.375975, -2.579052, -0.757362, 1.570796, 1.679603],accel_mss,speed_ms,0,blend_radius_m)
    |   movel([0.109317, -1.375221, -2.579578, -0.757590, 1.570796, 1.680113],accel_mss,speed_ms,0,blend_radius_m)
    |   movel([0.110409, -1.374305, -2.580215, -0.757869, 1.570796, 1.681205],accel_mss,speed_ms,0,blend_radius_m)
    |   movel([0.111301, -1.373912, -2.580489, -0.757989, 1.570796, 1.682097],accel_mss,speed_ms,0,blend_radius_m)
    |   movel([0.112411, -1.373819, -2.580553, -0.758017, 1.570796, 1.683208],accel_mss,speed_ms,0,blend_radius_m)
    |   movel([0.113017, -1.374036, -2.580403, -0.757951, 1.570796, 1.683814],accel_mss,speed_ms,0,blend_radius_m)
    |   movel([0.113017, -1.352274, -2.570239, -0.789876, 1.570796, 1.683814],accel_mss,speed_ms,0,blend_radius_m)
    |   movel([0.092010, -1.359781, -2.565150, -0.787458, 1.570796, 1.662807],accel_mss,speed_ms,0,blend_radius_m)
    |   movel([0.092010, -1.381418, -2.575232, -0.755739, 1.570796, 1.662807],accel_mss,speed_ms,0,blend_radius_m)
    |   movel([0.091844, -1.382062, -2.574777, -0.755550, 1.570796, 1.662640],accel_mss,speed_ms,0,blend_radius_m)
    |   movel([0.091053, -1.383210, -2.573965, -0.755214, 1.570796, 1.661849],accel_mss,speed_ms,0,blend_radius_m)
    |   movel([0.090244, -1.383849, -2.573512, -0.755028, 1.570796, 1.661040],accel_mss,speed_ms,0,blend_radius_m)
    |   movel([0.089338, -1.384266, -2.573216, -0.754907, 1.570796, 1.660134],accel_mss,speed_ms,0,blend_radius_m)
    |   movel([0.087854, -1.384288, -2.573201, -0.754900, 1.570796, 1.658650],accel_mss,speed_ms,0,blend_radius_m)
    |   movel([0.087133, -1.383609, -2.573682, -0.755097, 1.570796, 1.657929],accel_mss,speed_ms,0,blend_radius_m)
    |   movel([0.087027, -1.382857, -2.574215, -0.755317, 1.570796, 1.657823],accel_mss,speed_ms,0,blend_radius_m)
    |   movel([0.087252, -1.382080, -2.574764, -0.755544, 1.570796, 1.658048],accel_mss,speed_ms,0,blend_radius_m)
    |   movel([0.087730, -1.381334, -2.575291, -0.755764, 1.570796, 1.658527],accel_mss,speed_ms,0,blend_radius_m)
    |   movel([0.088813, -1.380412, -2.575942, -0.756036, 1.570796, 1.659610],accel_mss,speed_ms,0,blend_radius_m)
    |   movel([0.089697, -1.380008, -2.576225, -0.756155, 1.570796, 1.660494],accel_mss,speed_ms,0,blend_radius_m)
    |   movel([0.090807, -1.379897, -2.576304, -0.756188, 1.570796, 1.661604],accel_mss,speed_ms,0,blend_radius_m)
    |   movel([0.091420, -1.380098, -2.576162, -0.756129, 1.570796, 1.662217],accel_mss,speed_ms,0,blend_radius_m)
    |   movel([0.091954, -1.380805, -2.575665, -0.755920, 1.570796, 1.662751],accel_mss,speed_ms,0,blend_radius_m)
    |   movel([0.092010, -1.381418, -2.575232, -0.755739, 1.570796, 1.662807],accel_mss,speed_ms,0,blend_radius_m)
    |   movel([0.091844, -1.382062, -2.574777, -0.755550, 1.570796, 1.662640],accel_mss,speed_ms,0,blend_radius_m)
    |   movel([0.091053, -1.383210, -2.573965, -0.755214, 1.570796, 1.661849],accel_mss,speed_ms,0,blend_radius_m)
    |   movel([0.090244, -1.383849, -2.573512, -0.755028, 1.570796, 1.661040],accel_mss,speed_ms,0,blend_radius_m)
    |   movel([0.089338, -1.384266, -2.573216, -0.754907, 1.570796, 1.660134],accel_mss,speed_ms,0,blend_radius_m)
    |   movel([0.087854, -1.384288, -2.573201, -0.754900, 1.570796, 1.658650],accel_mss,speed_ms,0,blend_radius_m)
    |   movel([0.087133, -1.383609, -2.573682, -0.755097, 1.570796, 1.657929],accel_mss,speed_ms,0,blend_radius_m)
    |   movel([0.087027, -1.382857, -2.574215, -0.755317, 1.570796, 1.657823],accel_mss,speed_ms,0,blend_radius_m)
    |   movel([0.087252, -1.382080, -2.574764, -0.755544, 1.570796, 1.658048],accel_mss,speed_ms,0,blend_radius_m)
    |   movel([0.087730, -1.381334, -2.575291, -0.755764, 1.570796, 1.658527],accel_mss,speed_ms,0,blend_radius_m)
    |   movel([0.088813, -1.380412, -2.575942, -0.756036, 1.570796, 1.659610],accel_mss,speed_ms,0,blend_radius_m)
    |   movel([0.089697, -1.380008, -2.576225, -0.756155, 1.570796, 1.660494],accel_mss,speed_ms,0,blend_radius_m)
    |   movel([0.090807, -1.379897, -2.576304, -0.756188, 1.570796, 1.661604],accel_mss,speed_ms,0,blend_radius_m)
    |   movel([0.091420, -1.380098, -2.576162, -0.756129, 1.570796, 1.662217],accel_mss,speed_ms,0,blend_radius_m)
    |   movel([0.091954, -1.380805, -2.575665, -0.755920, 1.570796, 1.662751],accel_mss,speed_ms,0,blend_radius_m)
    |   movel([0.092010, -1.381418, -2.575232, -0.755739, 1.570796, 1.662807],accel_mss,speed_ms,0,blend_radius_m)
    |   movel([0.092010, -1.359781, -2.565150, -0.787458, 1.570796, 1.662807],accel_mss,speed_ms,0,blend_radius_m)
    |   movel([0.094674, -1.359006, -2.565679, -0.787704, 1.570796, 1.665471],accel_mss,speed_ms,0,blend_radius_m)
    |   movel([0.094674, -1.380655, -2.575770, -0.755964, 1.570796, 1.665471],accel_mss,speed_ms,0,blend_radius_m)
    |   movel([0.094322, -1.381982, -2.574834, -0.755573, 1.570796, 1.665118],accel_mss,speed_ms,0,blend_radius_m)
    |   movel([0.092703, -1.384356, -2.573152, -0.754880, 1.570796, 1.663499],accel_mss,speed_ms,0,blend_radius_m)
    |   movel([0.091021, -1.385680, -2.572211, -0.754498, 1.570796, 1.661817],accel_mss,speed_ms,0,blend_radius_m)
    |   movel([0.089151, -1.386528, -2.571607, -0.754254, 1.570796, 1.659947],accel_mss,speed_ms,0,blend_radius_m)
    |   movel([0.086092, -1.386578, -2.571572, -0.754240, 1.570796, 1.656888],accel_mss,speed_ms,0,blend_radius_m)
    |   movel([0.084580, -1.385186, -2.572563, -0.754640, 1.570796, 1.655376],accel_mss,speed_ms,0,blend_radius_m)
    |   movel([0.084368, -1.383631, -2.573667, -0.755091, 1.570796, 1.655165],accel_mss,speed_ms,0,blend_radius_m)
    |   movel([0.084831, -1.382033, -2.574798, -0.755558, 1.570796, 1.655627],accel_mss,speed_ms,0,blend_radius_m)
    |   movel([0.085815, -1.380489, -2.575887, -0.756013, 1.570796, 1.656611],accel_mss,speed_ms,0,blend_radius_m)
    |   movel([0.088052, -1.378554, -2.577248, -0.756588, 1.570796, 1.658849],accel_mss,speed_ms,0,blend_radius_m)
    |   movel([0.089888, -1.377724, -2.577829, -0.756836, 1.570796, 1.660684],accel_mss,speed_ms,0,blend_radius_m)
    |   movel([0.092200, -1.377486, -2.577996, -0.756907, 1.570796, 1.662997],accel_mss,speed_ms,0,blend_radius_m)
    |   movel([0.093462, -1.377912, -2.577697, -0.756780, 1.570796, 1.664259],accel_mss,speed_ms,0,blend_radius_m)
    |   movel([0.094572, -1.379372, -2.576673, -0.756344, 1.570796, 1.665368],accel_mss,speed_ms,0,blend_radius_m)
    |   movel([0.094674, -1.380655, -2.575770, -0.755964, 1.570796, 1.665471],accel_mss,speed_ms,0,blend_radius_m)
    |   movel([0.094322, -1.381982, -2.574834, -0.755573, 1.570796, 1.665118],accel_mss,speed_ms,0,blend_radius_m)
    |   movel([0.092703, -1.384356, -2.573152, -0.754880, 1.570796, 1.663499],accel_mss,speed_ms,0,blend_radius_m)
    |   movel([0.091021, -1.385680, -2.572211, -0.754498, 1.570796, 1.661817],accel_mss,speed_ms,0,blend_radius_m)
    |   movel([0.089151, -1.386528, -2.571607, -0.754254, 1.570796, 1.659947],accel_mss,speed_ms,0,blend_radius_m)
    |   movel([0.086092, -1.386578, -2.571572, -0.754240, 1.570796, 1.656888],accel_mss,speed_ms,0,blend_radius_m)
    |   movel([0.084580, -1.385186, -2.572563, -0.754640, 1.570796, 1.655376],accel_mss,speed_ms,0,blend_radius_m)
    |   movel([0.084368, -1.383631, -2.573667, -0.755091, 1.570796, 1.655165],accel_mss,speed_ms,0,blend_radius_m)
    |   movel([0.084831, -1.382033, -2.574798, -0.755558, 1.570796, 1.655627],accel_mss,speed_ms,0,blend_radius_m)
    |   movel([0.085815, -1.380489, -2.575887, -0.756013, 1.570796, 1.656611],accel_mss,speed_ms,0,blend_radius_m)
    |   movel([0.088052, -1.378554, -2.577248, -0.756588, 1.570796, 1.658849],accel_mss,speed_ms,0,blend_radius_m)
    |   movel([0.089888, -1.377724, -2.577829, -0.756836, 1.570796, 1.660684],accel_mss,speed_ms,0,blend_radius_m)
    |   movel([0.092200, -1.377486, -2.577996, -0.756907, 1.570796, 1.662997],accel_mss,speed_ms,0,blend_radius_m)
    |   movel([0.093462, -1.377912, -2.577697, -0.756780, 1.570796, 1.664259],accel_mss,speed_ms,0,blend_radius_m)
    |   movel([0.094572, -1.379372, -2.576673, -0.756344, 1.570796, 1.665368],accel_mss,speed_ms,0,blend_radius_m)
    |   movel([0.094674, -1.380655, -2.575770, -0.755964, 1.570796, 1.665471],accel_mss,speed_ms,0,blend_radius_m)
    |   movel([0.094674, -1.359006, -2.565679, -0.787704, 1.570796, 1.665471],accel_mss,speed_ms,0,blend_radius_m)
    |   movel([0.092538, -1.346767, -2.573922, -0.791699, 1.570796, 1.663334],accel_mss,speed_ms,0,blend_radius_m)
    |   movel([0.092538, -1.368619, -2.584146, -0.759623, 1.570796, 1.663334],accel_mss,speed_ms,0,blend_radius_m)
    |   movel([0.089149, -1.370309, -2.582983, -0.759097, 1.570796, 1.659945],accel_mss,speed_ms,0,blend_radius_m)
    |   movel([0.089391, -1.368693, -2.584096, -0.759600, 1.570796, 1.660187],accel_mss,speed_ms,0,blend_radius_m)
    |   movel([0.092287, -1.367155, -2.585151, -0.760083, 1.570796, 1.663083],accel_mss,speed_ms,0,blend_radius_m)
    |   movel([0.098130, -1.364590, -2.586904, -0.760895, 1.570796, 1.668926],accel_mss,speed_ms,0,blend_radius_m)
    |   movel([0.101754, -1.363359, -2.587742, -0.761288, 1.570796, 1.672550],accel_mss,speed_ms,0,blend_radius_m)
    |   movel([0.104529, -1.362638, -2.588232, -0.761519, 1.570796, 1.675325],accel_mss,speed_ms,0,blend_radius_m)
    |   movel([0.107614, -1.362028, -2.588646, -0.761715, 1.570796, 1.678410],accel_mss,speed_ms,0,blend_radius_m)
    |   movel([0.110821, -1.361629, -2.588917, -0.761844, 1.570796, 1.681618],accel_mss,speed_ms,0,blend_radius_m)
    |   movel([0.114490, -1.361488, -2.589012, -0.761889, 1.570796, 1.685286],accel_mss,speed_ms,0,blend_radius_m)
    |   movel([0.114278, -1.363101, -2.587918, -0.761370, 1.570796, 1.685074],accel_mss,speed_ms,0,blend_radius_m)
    |   movel([0.110187, -1.363403, -2.587712, -0.761273, 1.570796, 1.680984],accel_mss,speed_ms,0,blend_radius_m)
    |   movel([0.107097, -1.363898, -2.587376, -0.761115, 1.570796, 1.677894],accel_mss,speed_ms,0,blend_radius_m)
    |   movel([0.104159, -1.364572, -2.586916, -0.760900, 1.570796, 1.674956],accel_mss,speed_ms,0,blend_radius_m)
    |   movel([0.101524, -1.365316, -2.586409, -0.760664, 1.570796, 1.672320],accel_mss,speed_ms,0,blend_radius_m)
    |   movel([0.098101, -1.366368, -2.585690, -0.760331, 1.570796, 1.668898],accel_mss,speed_ms,0,blend_radius_m)
    |   movel([0.092538, -1.368619, -2.584146, -0.759623, 1.570796, 1.663334],accel_mss,speed_ms,0,blend_radius_m)
    |   movel([0.089149, -1.370309, -2.582983, -0.759097, 1.570796, 1.659945],accel_mss,speed_ms,0,blend_radius_m)
    |   movel([0.089391, -1.368693, -2.584096, -0.759600, 1.570796, 1.660187],accel_mss,speed_ms,0,blend_radius_m)
    |   movel([0.092287, -1.367155, -2.585151, -0.760083, 1.570796, 1.663083],accel_mss,speed_ms,0,blend_radius_m)
    |   movel([0.098130, -1.364590, -2.586904, -0.760895, 1.570796, 1.668926],accel_mss,speed_ms,0,blend_radius_m)
    |   movel([0.101754, -1.363359, -2.587742, -0.761288, 1.570796, 1.672550],accel_mss,speed_ms,0,blend_radius_m)
    |   movel([0.104529, -1.362638, -2.588232, -0.761519, 1.570796, 1.675325],accel_mss,speed_ms,0,blend_radius_m)
    |   movel([0.107614, -1.362028, -2.588646, -0.761715, 1.570796, 1.678410],accel_mss,speed_ms,0,blend_radius_m)
    |   movel([0.110821, -1.361629, -2.588917, -0.761844, 1.570796, 1.681618],accel_mss,speed_ms,0,blend_radius_m)
    |   movel([0.114490, -1.361488, -2.589012, -0.761889, 1.570796, 1.685286],accel_mss,speed_ms,0,blend_radius_m)
    |   movel([0.114278, -1.363101, -2.587918, -0.761370, 1.570796, 1.685074],accel_mss,speed_ms,0,blend_radius_m)
    |   movel([0.110187, -1.363403, -2.587712, -0.761273, 1.570796, 1.680984],accel_mss,speed_ms,0,blend_radius_m)
    |   movel([0.107097, -1.363898, -2.587376, -0.761115, 1.570796, 1.677894],accel_mss,speed_ms,0,blend_radius_m)
    |   movel([0.104159, -1.364572, -2.586916, -0.760900, 1.570796, 1.674956],accel_mss,speed_ms,0,blend_radius_m)
    |   movel([0.101524, -1.365316, -2.586409, -0.760664, 1.570796, 1.672320],accel_mss,speed_ms,0,blend_radius_m)
    |   movel([0.098101, -1.366368, -2.585690, -0.760331, 1.570796, 1.668898],accel_mss,speed_ms,0,blend_radius_m)
    |   movel([0.092538, -1.368619, -2.584146, -0.759623, 1.570796, 1.663334],accel_mss,speed_ms,0,blend_radius_m)
    |   movel([0.092538, -1.346767, -2.573922, -0.791699, 1.570796, 1.663334],accel_mss,speed_ms,0,blend_radius_m)
    |   movel([0.076452, -1.354004, -2.569073, -0.789312, 1.570796, 1.647248],accel_mss,speed_ms,0,blend_radius_m)
    |   movel([0.076452, -1.375736, -2.579218, -0.757434, 1.570796, 1.647248],accel_mss,speed_ms,0,blend_radius_m)
    |   movel([0.075395, -1.387611, -2.570834, -0.753944, 1.570796, 1.646191],accel_mss,speed_ms,0,blend_radius_m)
    |   movel([0.074759, -1.388898, -2.569913, -0.753578, 1.570796, 1.645555],accel_mss,speed_ms,0,blend_radius_m)
    |   movel([0.073372, -1.389777, -2.569282, -0.753329, 1.570796, 1.644168],accel_mss,speed_ms,0,blend_radius_m)
    |   movel([0.072266, -1.389798, -2.569268, -0.753324, 1.570796, 1.643062],accel_mss,speed_ms,0,blend_radius_m)
    |   movel([0.071627, -1.388738, -2.570028, -0.753623, 1.570796, 1.642423],accel_mss,speed_ms,0,blend_radius_m)
    |   movel([0.072629, -1.376899, -2.578406, -0.757084, 1.570796, 1.643426],accel_mss,speed_ms,0,blend_radius_m)
    |   movel([0.073422, -1.375424, -2.579436, -0.757529, 1.570796, 1.644218],accel_mss,speed_ms,0,blend_radius_m)
    |   movel([0.074684, -1.374669, -2.579962, -0.757758, 1.570796, 1.645480],accel_mss,speed_ms,0,blend_radius_m)
    |   movel([0.075652, -1.374607, -2.580005, -0.757777, 1.570796, 1.646449],accel_mss,speed_ms,0,blend_radius_m)
    |   movel([0.076452, -1.375736, -2.579218, -0.757434, 1.570796, 1.647248],accel_mss,speed_ms,0,blend_radius_m)
    |   movel([0.075395, -1.387611, -2.570834, -0.753944, 1.570796, 1.646191],accel_mss,speed_ms,0,blend_radius_m)
    |   movel([0.074759, -1.388898, -2.569913, -0.753578, 1.570796, 1.645555],accel_mss,speed_ms,0,blend_radius_m)
    |   movel([0.073372, -1.389777, -2.569282, -0.753329, 1.570796, 1.644168],accel_mss,speed_ms,0,blend_radius_m)
    |   movel([0.072266, -1.389798, -2.569268, -0.753324, 1.570796, 1.643062],accel_mss,speed_ms,0,blend_radius_m)
    |   movel([0.071627, -1.388738, -2.570028, -0.753623, 1.570796, 1.642423],accel_mss,speed_ms,0,blend_radius_m)
    |   movel([0.072629, -1.376899, -2.578406, -0.757084, 1.570796, 1.643426],accel_mss,speed_ms,0,blend_radius_m)
    |   movel([0.073422, -1.375424, -2.579436, -0.757529, 1.570796, 1.644218],accel_mss,speed_ms,0,blend_radius_m)
    |   movel([0.074684, -1.374669, -2.579962, -0.757758, 1.570796, 1.645480],accel_mss,speed_ms,0,blend_radius_m)
    |   movel([0.075652, -1.374607, -2.580005, -0.757777, 1.570796, 1.646449],accel_mss,speed_ms,0,blend_radius_m)
    |   movel([0.076452, -1.375736, -2.579218, -0.757434, 1.570796, 1.647248],accel_mss,speed_ms,0,blend_radius_m)
    |   movel([0.076452, -1.354004, -2.569073, -0.789312, 1.570796, 1.647248],accel_mss,speed_ms,0,blend_radius_m)
    |   movel([0.077651, -1.340455, -2.578095, -0.793839, 1.570796, 1.648448],accel_mss,speed_ms,0,blend_radius_m)
    |   movel([0.077651, -1.362409, -2.588387, -0.761592, 1.570796, 1.648448],accel_mss,speed_ms,0,blend_radius_m)
    |   movel([0.078010, -1.361212, -2.589199, -0.761978, 1.570796, 1.648807],accel_mss,speed_ms,0,blend_radius_m)
    |   movel([0.080092, -1.359026, -2.590675, -0.762688, 1.570796, 1.650888],accel_mss,speed_ms,0,blend_radius_m)
    |   movel([0.081259, -1.358494, -2.591034, -0.762862, 1.570796, 1.652055],accel_mss,speed_ms,0,blend_radius_m)
    |   movel([0.125839, -1.345452, -2.599692, -0.767245, 1.570796, 1.696635],accel_mss,speed_ms,0,blend_radius_m)
    |   movel([0.127075, -1.345321, -2.599778, -0.767290, 1.570796, 1.697871],accel_mss,speed_ms,0,blend_radius_m)
    |   movel([0.128721, -1.346495, -2.599009, -0.766886, 1.570796, 1.699518],accel_mss,speed_ms,0,blend_radius_m)
    |   movel([0.128784, -1.347516, -2.598338, -0.766535, 1.570796, 1.699581],accel_mss,speed_ms,0,blend_radius_m)
    |   movel([0.123841, -1.381676, -2.575050, -0.755663, 1.570796, 1.694637],accel_mss,speed_ms,0,blend_radius_m)
    |   movel([0.123467, -1.382782, -2.574268, -0.755339, 1.570796, 1.694263],accel_mss,speed_ms,0,blend_radius_m)
    |   movel([0.121776, -1.384615, -2.572968, -0.754805, 1.570796, 1.692573],accel_mss,speed_ms,0,blend_radius_m)
    |   movel([0.120210, -1.385338, -2.572455, -0.754596, 1.570796, 1.691006],accel_mss,speed_ms,0,blend_radius_m)
    |   movel([0.077671, -1.397098, -2.563988, -0.751303, 1.570796, 1.648468],accel_mss,speed_ms,0,blend_radius_m)
    |   movel([0.076660, -1.397250, -2.563878, -0.751261, 1.570796, 1.647457],accel_mss,speed_ms,0,blend_radius_m)
    |   movel([0.074964, -1.396457, -2.564455, -0.751477, 1.570796, 1.645760],accel_mss,speed_ms,0,blend_radius_m)
    |   movel([0.074716, -1.395310, -2.565289, -0.751790, 1.570796, 1.645512],accel_mss,speed_ms,0,blend_radius_m)
    |   movel([0.077651, -1.362409, -2.588387, -0.761592, 1.570796, 1.648448],accel_mss,speed_ms,0,blend_radius_m)
    |   movel([0.078010, -1.361212, -2.589199, -0.761978, 1.570796, 1.648807],accel_mss,speed_ms,0,blend_radius_m)
    |   movel([0.080092, -1.359026, -2.590675, -0.762688, 1.570796, 1.650888],accel_mss,speed_ms,0,blend_radius_m)
    |   movel([0.081259, -1.358494, -2.591034, -0.762862, 1.570796, 1.652055],accel_mss,speed_ms,0,blend_radius_m)
    |   movel([0.125839, -1.345452, -2.599692, -0.767245, 1.570796, 1.696635],accel_mss,speed_ms,0,blend_radius_m)
    |   movel([0.127075, -1.345321, -2.599778, -0.767290, 1.570796, 1.697871],accel_mss,speed_ms,0,blend_radius_m)
    |   movel([0.128721, -1.346495, -2.599009, -0.766886, 1.570796, 1.699518],accel_mss,speed_ms,0,blend_radius_m)
    |   movel([0.128784, -1.347516, -2.598338, -0.766535, 1.570796, 1.699581],accel_mss,speed_ms,0,blend_radius_m)
    |   movel([0.123841, -1.381676, -2.575050, -0.755663, 1.570796, 1.694637],accel_mss,speed_ms,0,blend_radius_m)
    |   movel([0.123467, -1.382782, -2.574268, -0.755339, 1.570796, 1.694263],accel_mss,speed_ms,0,blend_radius_m)
    |   movel([0.121776, -1.384615, -2.572968, -0.754805, 1.570796, 1.692573],accel_mss,speed_ms,0,blend_radius_m)
    |   movel([0.120210, -1.385338, -2.572455, -0.754596, 1.570796, 1.691006],accel_mss,speed_ms,0,blend_radius_m)
    |   movel([0.077671, -1.397098, -2.563988, -0.751303, 1.570796, 1.648468],accel_mss,speed_ms,0,blend_radius_m)
    |   movel([0.076660, -1.397250, -2.563878, -0.751261, 1.570796, 1.647457],accel_mss,speed_ms,0,blend_radius_m)
    |   movel([0.074964, -1.396457, -2.564455, -0.751477, 1.570796, 1.645760],accel_mss,speed_ms,0,blend_radius_m)
    |   movel([0.074716, -1.395310, -2.565289, -0.751790, 1.570796, 1.645512],accel_mss,speed_ms,0,blend_radius_m)
    |   movel([0.077651, -1.362409, -2.588387, -0.761592, 1.570796, 1.648448],accel_mss,speed_ms,0,blend_radius_m)
    |   movel([0.077651, -1.340455, -2.578095, -0.793839, 1.570796, 1.648448],accel_mss,speed_ms,0,blend_radius_m)
    |   movel([0.070954, -1.327862, -2.586258, -0.798269, 1.570796, 1.641750],accel_mss,speed_ms,0,blend_radius_m)
    |   movel([0.070954, -1.350017, -2.596688, -0.765684, 1.570796, 1.641750],accel_mss,speed_ms,0,blend_radius_m)
    |   movel([0.053570, -1.353872, -2.594129, -0.764388, 1.570796, 1.624367],accel_mss,speed_ms,0,blend_radius_m)
    |   movel([0.070954, -1.350017, -2.596688, -0.765684, 1.570796, 1.641750],accel_mss,speed_ms,0,blend_radius_m)
    |   movel([0.070954, -1.327862, -2.586258, -0.798269, 1.570796, 1.641750],accel_mss,speed_ms,0,blend_radius_m)
    |   movel([0.051927, -1.332380, -2.583353, -0.796655, 1.570796, 1.622724],accel_mss,speed_ms,0,blend_radius_m)
    |   movel([0.051927, -1.354464, -2.593734, -0.764191, 1.570796, 1.622724],accel_mss,speed_ms,0,blend_radius_m)
    |   movel([0.072897, -1.350052, -2.596665, -0.765672, 1.570796, 1.643693],accel_mss,speed_ms,0,blend_radius_m)
    |   movel([0.072268, -1.357488, -2.591709, -0.763191, 1.570796, 1.643064],accel_mss,speed_ms,0,blend_radius_m)
    |   movel([0.069919, -1.358610, -2.590955, -0.762824, 1.570796, 1.640715],accel_mss,speed_ms,0,blend_radius_m)
    |   movel([0.066289, -1.359896, -2.590089, -0.762405, 1.570796, 1.637085],accel_mss,speed_ms,0,blend_radius_m)
    |   movel([0.062781, -1.360622, -2.589598, -0.762169, 1.570796, 1.633578],accel_mss,speed_ms,0,blend_radius_m)
    |   movel([0.056737, -1.360442, -2.589720, -0.762227, 1.570796, 1.627533],accel_mss,speed_ms,0,blend_radius_m)
    |   movel([0.053559, -1.359310, -2.590483, -0.762595, 1.570796, 1.624355],accel_mss,speed_ms,0,blend_radius_m)
    |   movel([0.051925, -1.358255, -2.591194, -0.762940, 1.570796, 1.622721],accel_mss,speed_ms,0,blend_radius_m)
    |   movel([0.051927, -1.354464, -2.593734, -0.764191, 1.570796, 1.622724],accel_mss,speed_ms,0,blend_radius_m)
    |   movel([0.072897, -1.350052, -2.596665, -0.765672, 1.570796, 1.643693],accel_mss,speed_ms,0,blend_radius_m)
    |   movel([0.072268, -1.357488, -2.591709, -0.763191, 1.570796, 1.643064],accel_mss,speed_ms,0,blend_radius_m)
    |   movel([0.069919, -1.358610, -2.590955, -0.762824, 1.570796, 1.640715],accel_mss,speed_ms,0,blend_radius_m)
    |   movel([0.066289, -1.359896, -2.590089, -0.762405, 1.570796, 1.637085],accel_mss,speed_ms,0,blend_radius_m)
    |   movel([0.062781, -1.360622, -2.589598, -0.762169, 1.570796, 1.633578],accel_mss,speed_ms,0,blend_radius_m)
    |   movel([0.056737, -1.360442, -2.589720, -0.762227, 1.570796, 1.627533],accel_mss,speed_ms,0,blend_radius_m)
    |   movel([0.053559, -1.359310, -2.590483, -0.762595, 1.570796, 1.624355],accel_mss,speed_ms,0,blend_radius_m)
    |   movel([0.051925, -1.358255, -2.591194, -0.762940, 1.570796, 1.622721],accel_mss,speed_ms,0,blend_radius_m)
